// -------------------------------------------------
// Maintenance
      A     #U.Seq.Switch.Sw31;
      OPN   DB   500;
      =     DBX [AR2,P#0.0]; //"PStatD".U[#UnitNo].MTNC
// -------------------------------------------------
// CIP Required
// -------------------------------------------------
// CIP Active
// -------------------------------------------------
// CIP Clean
// -------------------------------------------------
// SIP Required
// -------------------------------------------------
// SIP Active
// -------------------------------------------------
// SIP Clean
// -------------------------------------------------
// Full
      A     DB135.DBX   26.2;
      OPN   DB   500;
      =     DBX [AR2,P#0.7]; //"PStatD".U[#UnitNo].FULL
// -------------------------------------------------
// Filling
      A     DB135.DBX   26.1;
      OPN   DB   500;
      =     DBX [AR2,P#1.0]; //"PStatD".U[#UnitNo].FILL
// -------------------------------------------------
// Ready For Filling
      A     DB135.DBX   26.0;
      OPN   DB   500;
      =     DBX [AR2,P#1.1]; //"PStatD".U[#UnitNo].RFFI
// -------------------------------------------------
// Empty
      A     DB135.DBX   26.5;
      OPN   DB   500;
      =     DBX [AR2,P#1.2]; //"PStatD".U[#UnitNo].EMTY
// -------------------------------------------------
// Emptying
      A     DB135.DBX   26.4;
      OPN   DB   500;
      =     DBX [AR2,P#1.3]; //"PStatD".U[#UnitNo].EMTI
// -------------------------------------------------
// Ready For Emptying
      A     DB135.DBX   26.3;
      OPN   DB   500;
      =     DBX [AR2,P#1.4]; //"PStatD".U[#UnitNo].RFEM
// -------------------------------------------------
// Reserved
//      A     #ComXYZ
//      OPN   "PStatD"
//      =     DBX [AR2,P#1.5]             //"PStatD".U[#UnitNo].RESV
// -------------------------------------------------
// Production
// -------------------------------------------------
// Used

// -------------------------------------------------
// PStat Function Call

      CALL FC   500 (
           UnitNo                   := #UnitNo,
           PStatModVal              := DB235.DBD  234);

NETWORK
TITLE =Unit Hold Request and Messages

      SET   ;

// ---------------------------------------------------------------------------
// Set unit to "hold" if maintenance
      AN    #U.Seq.Switch.Sw31; // maintenance !
      JC    NCO1;
      S     M    120.3;
      L     998; // "Unit in maintenance !"
      T     MD    90;

// ---------------------------------------------------------------------------
// Set unit to "hold" if emergency stop
NCO1: A     #EStopOK;
      JC    NCO2;
      S     M    120.3;
      L     999; // "Emergency stop !"
      T     MD    90;
NCO2: NOP   0;


// ---------------------------------------------------------------------------
// Check Partner
      AN    #ComSRC;
      O(    ;
      AN    DB135.DBX  314.3;
      AN    DB135.DBX  314.4;
      )     ;
      AN    #U.Seq.Step0;
      AN    #CIP;
      JCN   NC03;
      L     904; // "Source Not Ready!
      T     MD    90;
NC03: NOP   0;


      AN    DB135.DBX  266.0; // Water Tank Ready
      AN    DB135.DBX  266.1;
      AN    #ComDST;
      A     #S2I.SFM10.I00;
      AN    #U.Seq.Step0;
      AN    #U.Seq.PO.B22;
      AN    #U.Seq.PO.B3;
      AN    #CIP;
      JCN   NC04;
      L     903; // Destination not Ready
      T     MD    90;
NC04: NOP   0;



END_FUNCTION_BLOCK

FUNCTION_BLOCK FB 133
TITLE =C03: Local Well Transfer x
AUTHOR : Woermann
FAMILY : BOTEC_F1
NAME : C03E
VERSION : 1.2
CODE_VERSION1


VAR
  U : UDT 131;
END_VAR
VAR_TEMP
  CIP : BOOL ;	//CIP active
  UNIM : BOOL ;	//Unit Not In Maintenance
  GenRel : BOOL ;	//general OK (emergency and maintenance OK)
  EStopOK : BOOL ;	//emergency OK
  UnitNo : INT ;	//unit number
  xTmp : BOOL ;	//Temporary Bool
  iTmp : INT ;	//Temporary INT
  rTmp : REAL ;	//Temporary REAL
  dTmp : DINT ;	//Temporary DINT (free for general use)
  RetValInt : INT ;	//return value
  ComCIP1 : BOOL ;	//CIP1 in use
  ComCIP3 : BOOL ;	//CIP3 in use
END_VAR
BEGIN
NETWORK
TITLE =General

      SET   ;
// Simulation ---------------------------------------------------------------
      A     #U.Seq.User.Bit63;
      CC    FB   139; // "C03Sim"
      A     #U.Seq.Sim;
      =     #U.Seq.User.Bit63; //Help bit for simulation

// get unit number ----------------------------------------------------------
      L     MB   112;
      T     #UnitNo;

// CIP ----------------------------------------------------------------------
      L     #U.Seq.ProgNo;
      L     0;
      <D    ;
      =     #CIP;

// emergency OK -------------------------------------------------------------
      A     DB135.DBX   27.0; //Emergency Stop OK
      =     #EStopOK;

// Write Unit in Maintenance ------------------------------------------------

      AN    #U.Seq.Switch.Sw31;
      =     #UNIM;

// emergency and maintenance OK ---------------------------------------------
      A     #EStopOK;
      A     #UNIM;
      =     #GenRel;

// communication ------------------------------------------------------------
      UC    FB   135; // C03Com

NETWORK
TITLE =Analog Inputs

      NOP   0;

// ----------------------------------------------------------
// U31_AnI001 J6F_Druck
// ----------------------------------------------------------
      L     #U.Seq.SFM[63].Sp; // !!! insert correct SFM !!!
      T     DB233.DBD  238;

      SET   ;
      =     DB233.DBX  141.5;

// ----------------------------------------------------------
// QI_CO2_J6F_PH
// ----------------------------------------------------------
      L     #U.Seq.SFM[15].Sp;
      T     DB233.DBD  358;

      SET   ;
      =     DB233.DBX  261.5;

// ----------------------------------------------------------
// U31_AnI003 spare
// ----------------------------------------------------------
      L     #U.Seq.SFM[63].Sp; // !!! insert correct SFM !!!
      T     DB233.DBD  478;

      SET   ;
      =     DB233.DBX  381.5;

NETWORK
TITLE =Universal Value

      NOP   0;

// ----------------------------------------------------------
// unv001 Process Status
// ----------------------------------------------------------
// process value to UnV
//      L     0.000000e+000
//      T     "C03UnVD".unv001.ValExt

// ----------------------------------------------------------
// unv002 Universal Value 02
// ----------------------------------------------------------
// process value to UnV
//      L     0.000000e+000
//      T     "C03UnVD".unv002.ValExt

// ----------------------------------------------------------
// unv003 Universal Value 03
// ----------------------------------------------------------
// process value to UnV
//      L     0.000000e+000
//      T     "C03UnVD".unv003.ValExt

// ----------------------------------------------------------
// unv004 Universal Value 04
// ----------------------------------------------------------
// process value to UnV
//      L     0.000000e+000
//      T     "C03UnVD".unv004.ValExt

NETWORK
TITLE =Special Input

      NOP   0;

// ----------------------------------------------------------
// U31_SpI001 spare
// ----------------------------------------------------------
      CLR   ; // Only used in one well?
      =     DB231.DBX   81.4;
      =     DB231.DBX   81.5;

// ----------------------------------------------------------
// U31_SpI002 spare
// ----------------------------------------------------------
      CLR   ; // Only used in one well?
      =     DB231.DBX  141.4;
      =     DB231.DBX  141.5;

// ----------------------------------------------------------
// U31_SpI003 spare
// ----------------------------------------------------------
      CLR   ; // Only used in one well?
      =     DB231.DBX  201.4;
      =     DB231.DBX  201.5;

NETWORK
TITLE =Messages

      NOP   0;

// ----------------------------------------------------------
// msg001 Message 01
// ----------------------------------------------------------
      SET   ;
      R     DB237.DBX   80.7;
      =     DB237.DBX   81.4;

      CLR   ;
      =     DB237.DBX   82.7;

// ----------------------------------------------------------
// msg002 Message 02
// ----------------------------------------------------------
      SET   ;
      R     DB237.DBX  140.7;
      =     DB237.DBX  141.4;

      CLR   ;
      =     DB237.DBX  142.7;

// ----------------------------------------------------------
// msg003 Message 03
// ----------------------------------------------------------
      SET   ;
      R     DB237.DBX  200.7;
      =     DB237.DBX  201.4;

      CLR   ;
      =     DB237.DBX  202.7;

NETWORK
TITLE =PID controller
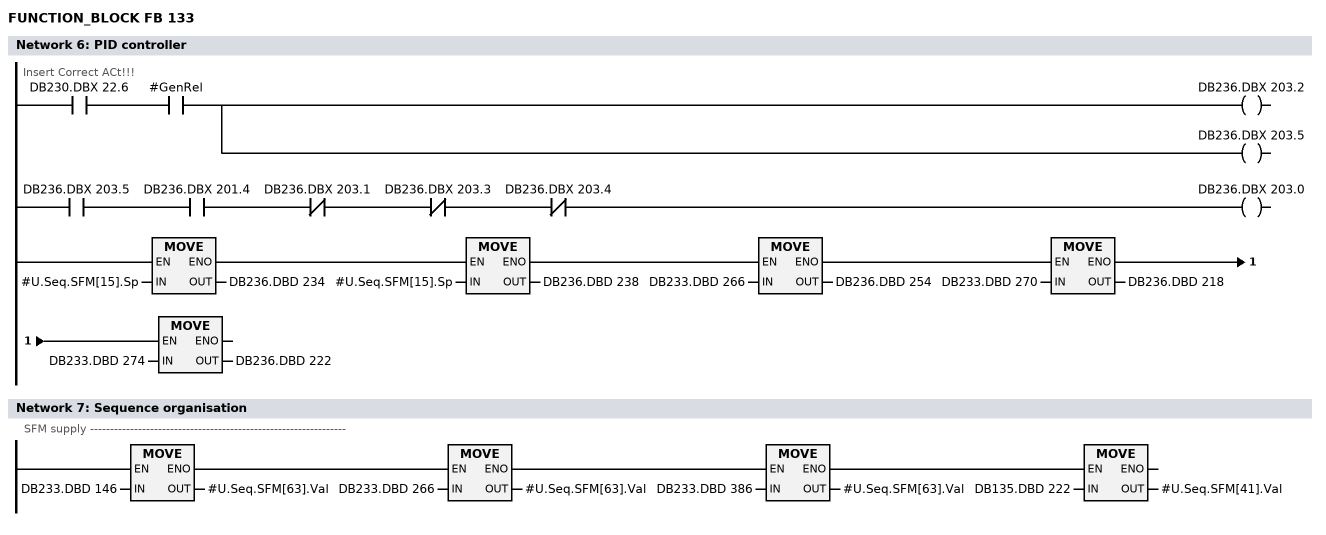

      NOP   0;

// ----------------------------------------------------------
// CO2J6FRV1 CO2 J6F RV1
// ----------------------------------------------------------
// starting value -----------------------
      A     DB230.DBX   22.6; // Insert Correct ACt!!!
      A     #GenRel;
      =     DB236.DBX  203.2;
      =     DB236.DBX  203.5;

// enable alarm -------------------------
      A     DB236.DBX  203.5;
      A     DB236.DBX  201.4;
      AN    DB236.DBX  203.1;
      AN    DB236.DBX  203.3;
      AN    DB236.DBX  203.4;
      =     DB236.DBX  203.0;

// setpoint to controller ---------------
      L     #U.Seq.SFM[15].Sp; // pH
      T     DB236.DBD  234;

// static value to controller ----------
      L     #U.Seq.SFM[15].Sp; //  pH
      T     DB236.DBD  238;

// process value to controller ----------
      L     DB233.DBD  266;
      T     DB236.DBD  254;

// low/high value to controller ---------
      L     DB233.DBD  270;
      T     DB236.DBD  218;

      L     DB233.DBD  274;
      T     DB236.DBD  222;

NETWORK
TITLE =Sequence organisation
//
// SFM supply ----------------------------------------------------------------

// analog value to SFM J6F_Druck -----------------------
      L     DB233.DBD  146;
      T     #U.Seq.SFM[63].Val;

// analog value to SFM QI_CO2_J6F_PH -------------------
      L     DB233.DBD  266;
      T     #U.Seq.SFM[63].Val; // !!! insert correct SFM !!!

// analog value to SFM spare -----------------------
      L     DB233.DBD  386;
      T     #U.Seq.SFM[63].Val; // !!! insert correct SFM !!!


// Amount from Well PLC04
      L     DB135.DBD  222;
      T     #U.Seq.SFM[41].Val;


NETWORK
TITLE =Auto / Manual

      SET   ;
      AN    M    122.2;
      JC    MODE;
      AN    M    120.1;

// assign actuator mode
      AN    M    120.1;
      =     DB230.DBX  105.4;
      =     DB230.DBX  185.4;
      =     DB230.DBX  265.4;

// assign PID mode
      S     DB236.DBX  201.4;
      S     DB236.DBX  201.5;

MODE: SET   ;

NETWORK
TITLE =C03_Act001 spare
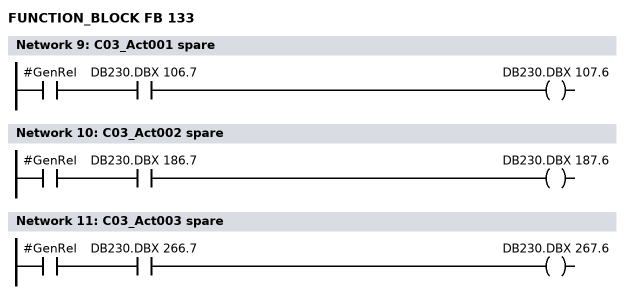

      A     #GenRel;
      A     DB230.DBX  106.7;
      =     DB230.DBX  107.6;
NETWORK
TITLE =C03_Act002 spare

      A     #GenRel;
      A     DB230.DBX  186.7;
      =     DB230.DBX  187.6;
NETWORK
TITLE =C03_Act003 spare

      A     #GenRel;
      A     DB230.DBX  266.7;
      =     DB230.DBX  267.6;
END_FUNCTION_BLOCK

FUNCTION_BLOCK FB 135
TITLE =C03: Local Well Transfer x
AUTHOR : Woermann
FAMILY : BOTEC_F1
NAME : C03Comm
VERSION : 0.1
CODE_VERSION1


VAR
  U : UDT 131;
END_VAR
VAR_TEMP
  iRetVal : INT ;	//return value as integer
  wRetVal : WORD ;	//return value as word
  Run : BOOL ;	//Unit in "RUN" mode
  EStopOK : BOOL ;	//Emergency Stop OK
  CIP : BOOL ;	//CIP Program Selected
  ComCIP : BOOL ;	//Communication with CIP Active
  xTmp : BOOL ;	//Temporary BOOL (free for general use)
  iTmp : INT ;	//Temporary INT (free for general use)
  rTmp : REAL ;	//Temporary REAL (free for general use)
  dTmp : DINT ;	//Temporary DINT (free for general use)
  UnitNo : INT ;	//Unit Number
  EquipmentID : INT ;	//Equipment ID
  Prid : DINT ;	//Process ID
  SFM36 : STRUCT 	//CIP Pump Mode
   I00 : BOOL ;	// Off
   I01 : BOOL ;	// Flow
   I02 : BOOL ;	// Pressure
   I03 : BOOL ;	// Fix Speed
   I04 : BOOL ;
   I05 : BOOL ;
   I06 : BOOL ;
   I07 : BOOL ;
   I08 : BOOL ;
   I09 : BOOL ;
   I10 : BOOL ;
   I11 : BOOL ;
   I12 : BOOL ;
   I13 : BOOL ;
   I14 : BOOL ;
   I15 : BOOL ;
   I16 : BOOL ;
   I17 : BOOL ;
   I18 : BOOL ;
   I19 : BOOL ;
   I20 : BOOL ;
   I21 : BOOL ;
   I22 : BOOL ;
   I23 : BOOL ;
   I24 : BOOL ;
   I25 : BOOL ;
   I26 : BOOL ;
   I27 : BOOL ;
   I28 : BOOL ;
   I29 : BOOL ;
   I30 : BOOL ;
   I31 : BOOL ;
  END_STRUCT ;
  iPLC : INT ;
  iUnit : INT ;
  rUnitNo : REAL ;
  DSTUnit : INT ;	//Destination Unit
END_VAR
BEGIN
NETWORK
TITLE =general

      SET   ;

// unit & equipment number ---------------------------------------------------
      L     #U.Seq.UnitNo;
      T     #UnitNo;

      L     DB135.DBW   14;
      L     1000;
      *I    ;
      L     #UnitNo;
      +I    ;
      T     #EquipmentID;

// CIP ----------------------------------------------------------------------
      L     DB135.DBW   18;
      L     0;
      <I    ;
      =     #CIP;

// Communicating Units-------------------------------------------------------
      L     DB135.DBD   10;
      L     DB135.DBD  106;
      ==D   ;
      =     #ComCIP;

// emergency OK -------------------------------------------------------------
      A     DB135.DBX   75.0; //General Emergency Stop OK
      =     #EStopOK;

NETWORK
TITLE =read other unit's data

      SET   ;

// ... General Unit ----------/
      CALL SFC   20 (
           SRCBLK                   := DB1995.Own,
           RET_VAL                  := #iTmp,
           DSTBLK                   := DB135.GEN);

// ... CIP Unit ------------- /

      CALL FC   563 (
           ActReq                   := M    101.0,
           PLCNo                    := 3,
           SourceUnitNo             := 91,
           IsTUnit                  := FALSE,
           DstComDRec               := DB135.CIP,
           RET_VAL                  := #wRetVal);

//----------------------------------------
// Communication Water Tank
//----------------------------------------
// Current Tank ----------------------------
      CALL FC   950 (
           EquipmentNo              := #U.Seq.SFM[10].Sp,
           PLCNo                    := #iPLC,
           UnitNo                   := #iUnit);

      L     #U.Seq.SFM[10].Sp;
      L     0.000000e+000;
      >R    ;
      JCN   N201;

      CALL FC   563 (
           ActReq                   := M    101.0,
           PLCNo                    := #iPLC,
           SourceUnitNo             := #iUnit,
           IsTUnit                  := FALSE,
           DstComDRec               := DB135.DST,
           RET_VAL                  := #wRetVal);
      JU    N2x1;
N201: NOP   0;
      L     0;
      T     #rTmp;
      CALL SFC   21 (
           BVAL                     := #rTmp,
           RET_VAL                  := #iTmp,
           BLK                      := DB135.DST);
N2x1: NOP   0;
// Priority 1 -----------------------------
      CALL FC   950 (
           EquipmentNo              := #U.Seq.SFM[11].Sp,
           PLCNo                    := #iPLC,
           UnitNo                   := #iUnit);

      L     #U.Seq.SFM[11].Sp;
      L     0.000000e+000;
      >R    ;
      JCN   N202;

      CALL FC   563 (
           ActReq                   := M    101.0,
           PLCNo                    := #iPLC,
           SourceUnitNo             := #iUnit,
           IsTUnit                  := FALSE,
           DstComDRec               := DB135.DST1,
           RET_VAL                  := #wRetVal);
      JU    N2x2;
N202: NOP   0;
      L     0;
      T     #rTmp;
      CALL SFC   21 (
           BVAL                     := #rTmp,
           RET_VAL                  := #iTmp,
           BLK                      := DB135.DST1);
N2x2: NOP   0;

// Priority 2 ----------------------------
      CALL FC   950 (
           EquipmentNo              := #U.Seq.SFM[12].Sp,
           PLCNo                    := #iPLC,
           UnitNo                   := #iUnit);

      L     #U.Seq.SFM[12].Sp;
      L     0.000000e+000;
      >R    ;
      JCN   N203;

      CALL FC   563 (
           ActReq                   := M    101.0,
           PLCNo                    := #iPLC,
           SourceUnitNo             := #iUnit,
           IsTUnit                  := FALSE,
           DstComDRec               := DB135.DST2,
           RET_VAL                  := #wRetVal);
      JU    N2x3;
N203: NOP   0;
      L     0;
      T     #rTmp;
      CALL SFC   21 (
           BVAL                     := #rTmp,
           RET_VAL                  := #iTmp,
           BLK                      := DB135.DST2);
N2x3: NOP   0;

// Priority 3 ----------------------------
      CALL FC   950 (
           EquipmentNo              := #U.Seq.SFM[13].Sp,
           PLCNo                    := #iPLC,
           UnitNo                   := #iUnit);

      L     #U.Seq.SFM[13].Sp;
      L     0.000000e+000;
      >R    ;
      JCN   N204;

      CALL FC   563 (
           ActReq                   := M    101.0,
           PLCNo                    := #iPLC,
           SourceUnitNo             := #iUnit,
           IsTUnit                  := FALSE,
           DstComDRec               := DB135.DST3,
           RET_VAL                  := #wRetVal);
      JU    N2x4;
N204: NOP   0;
      L     0;
      T     #rTmp;
      CALL SFC   21 (
           BVAL                     := #rTmp,
           RET_VAL                  := #iTmp,
           BLK                      := DB135.DST3);
N2x4: NOP   0;

//----------------------------------------
// Communication Water Treatment
//----------------------------------------
      L     21;
      L     DB135.DBW   16;
      ==I   ;
      JCN   WTR2;
      CALL FC   563 (
           ActReq                   := M    101.0,
           PLCNo                    := DB135.DBW   14,
           SourceUnitNo             := 38,
           IsTUnit                  := FALSE,
           DstComDRec               := DB135.PARTNER,
           RET_VAL                  := #wRetVal);
WTR2: L     22;
      ==I   ;
      JCN   NWTR;
      CALL FC   563 (
           ActReq                   := M    101.0,
           PLCNo                    := DB135.DBW   14,
           SourceUnitNo             := 39,
           IsTUnit                  := FALSE,
           DstComDRec               := DB135.PARTNER,
           RET_VAL                  := #wRetVal);

NWTR: NOP   0;

//----------------------------------------
// Communication Local Wells
//----------------------------------------
      L     #U.Seq.SFM[14].Sp; // Source
      T     #rTmp;

      CALL FC   950 (
           EquipmentNo              := #rTmp,
           PLCNo                    := #iPLC,
           UnitNo                   := #iUnit);

      L     #iUnit;
      L     1;
      ==I   ;
      JCN   U001;
      CALL SFC   20 (
           SRCBLK                   := DB1995.P04U001,
           RET_VAL                  := #iTmp,
           DSTBLK                   := DB135.SRC);
U001: NOP   0;

      L     #iUnit;
      L     2;
      ==I   ;
      JCN   U002;
      CALL SFC   20 (
           SRCBLK                   := DB1995.P04U002,
           RET_VAL                  := #iTmp,
           DSTBLK                   := DB135.SRC);
U002: NOP   0;

      L     #iUnit;
      L     3;
      ==I   ;
      JCN   U003;
      CALL SFC   20 (
           SRCBLK                   := DB1995.P04U003,
           RET_VAL                  := #iTmp,
           DSTBLK                   := DB135.SRC);
U003: NOP   0;

      L     #iUnit;
      L     4;
      ==I   ;
      JCN   U004;
      CALL SFC   20 (
           SRCBLK                   := DB1995.P04U004,
           RET_VAL                  := #iTmp,
           DSTBLK                   := DB135.SRC);
U004: NOP   0;

// Plan ----------------------------
      L     #UnitNo;
      L     100;
      +I    ;
      T     #iUnit;

      CALL FC   563 (
           ActReq                   := M    101.0,
           PLCNo                    := 3,
           SourceUnitNo             := #iUnit,
           IsTUnit                  := FALSE,
           DstComDRec               := DB135.PLN,
           RET_VAL                  := #wRetVal);

NETWORK
TITLE =external releases

      SET   ;
      =     DB230.DBX  106.7;
      =     DB230.DBX  186.7;
      =     DB230.DBX  266.7;

NETWORK
TITLE =write own unit data

      SET   ;
//-- CIP Communication ---------------------------------------
      AN    #U.Seq.Step0;
      AN    #U.Seq.PO.B30; // CIP Active (Slave)
      A     #ComCIP;
      JCN   NCIP;
//Conductivity CIP Return
      L     DB135.DBD  150;
      T     #U.Seq.SFM[32].Val;

//Temperature CIP Return
      L     DB135.DBD  146;
      T     #U.Seq.SFM[30].Val;

//CIP Prerun Pump SP

      CALL FC    45 (
           SFM                      := #U.Seq.SFM[36].Sp,
           Indexes                  := #SFM36);


      L     0.000000e+000;
      A     #SFM36.I01;
      =     DB135.DBX  171.7;
      JCN   pfc;
      L     #U.Seq.SFM[34].Sp;
pfc:  NOP   0;
      A     #SFM36.I02;
      =     DB135.DBX  172.0;
      JCN   ppc;
      L     #U.Seq.SFM[35].Sp;
ppc:  NOP   0;
      A     #SFM36.I03;
      =     DB135.DBX  171.6;
      JCN   pxc;
      L     #U.Seq.SFM[29].Sp;
pxc:  NOP   0;
      T     DB135.DBD  182;

//CIP Return
      L     #U.Seq.SFM[28].Sp;
      T     DB135.DBD  186;
      L     DB135.DBD  138;
      T     #U.Seq.SFM[28].Val;

//CIP Prerun
      L     #U.Seq.SFM[27].Sp;
      T     DB135.DBD  190;
      L     DB135.DBD  142;
      T     #U.Seq.SFM[27].Val;

// Write Own Data to CIP
      L     DB135.DBD   10;
      T     DB135.DBD  154;

      L     DB135.DBW   14;
      T     DB135.DBW  158;

      L     DB135.DBW   16;
      T     DB135.DBW  160;

      L     DB135.DBW   18;
      T     DB135.DBW  162;

      L     DB135.DBW   20;
      T     DB135.DBW  164;

      L     DB135.DBW   22;
      T     DB135.DBW  166;

      A     DB135.DBX   24.0;
      =     DB135.DBX  168.0;

      A     DB135.DBX   24.1;
      =     DB135.DBX  168.1;

      A     DB135.DBX   24.2;
      =     DB135.DBX  168.2;

      A     DB135.DBX   24.3;
      =     DB135.DBX  168.3;

      A     DB135.DBX   24.4;
      =     DB135.DBX  168.4;

      A     DB135.DBX   24.5;
      =     DB135.DBX  168.5;

      A     DB135.DBX   24.6;
      =     DB135.DBX  168.6;

      A     DB135.DBX   24.7;
      =     DB135.DBX  168.7;

// Copy Data to CIP
      CALL SFC   20 (
           SRCBLK                   := DB135.ToCIP,
           RET_VAL                  := #iRetVal,
           DSTBLK                   := DB135.ToCIP);

NCIP: NOP   0;

//Empty Signal
//A     "C03SpID".SpI.Sig //!!!! Insert correct Empty Signal !!!
      CLR   ;
      =     DB135.DBX   26.5;

//Full Signal
//A     "C03SpID".SpI.Sig //!!!! Insert correct Full Signal !!!
      CLR   ;
      =     DB135.DBX   26.2;

//CIP Program Selected
      A     #CIP;
      =     DB135.DBX   27.1;

// Emergency Stop
      A     #EStopOK; //If needed add or replace with own SpI
      =     DB135.DBX   27.0; //Emergency Stop OK

      L     #U.Seq.SFM[42].Sp; // Material
      T     DB135.DBD   30;

      L     DB135.DBD  326;
      T     #U.Seq.User.Real3;

//----------------------------------------
// Communication Water Tank
//----------------------------------------


      L     #U.Seq.SFM[10].Sp; // Current Tank
      T     DB135.DBD   34;

      L     #U.Seq.SFM[11].Sp; // Tank Priority 1
      T     DB135.DBD   38;

      L     #U.Seq.SFM[12].Sp; // Tank Priority 2
      T     DB135.DBD   42;

      L     #U.Seq.SFM[13].Sp; // Tank Priority 3
      T     DB135.DBD   46;

      L     #U.Seq.SFM[14].Sp; // Source
      T     DB135.DBD   50;

NETWORK
TITLE = read from other unit data




END_FUNCTION_BLOCK

FUNCTION_BLOCK FB 139
TITLE =C03: Local Well Transfer x
AUTHOR : Woermann
FAMILY : BOTEC_F1
NAME : C03Sim
VERSION : 0.1
CODE_VERSION1


VAR
  U : UDT 131;
END_VAR
VAR_TEMP
  CIP : BOOL ;	//CIP active
  xTmp : BOOL ;	//Temporary BOOL (free for general use)
  iTmp : INT ;	//Temporary INT (free for general use)
  rTmp : REAL ;	//Temporary REAL (free for general use)
  UnitNo : INT ;	//Unit Number
END_VAR
BEGIN
NETWORK
TITLE =General

      SET   ;
// get unit number ----------------------------------------------------------
      L     #U.Seq.UnitNo;
      T     #UnitNo;

// CIP ----------------------------------------------------------------------
      L     MW   114;
      L     0;
      <D    ;
      =     #CIP;

NETWORK
TITLE =Actuator

      A     #U.Seq.Sim;
      =     DB230.DBX  105.3;
      =     DB230.DBX  185.3;
      =     DB230.DBX  265.3;


NETWORK
TITLE =Special Input

      A     #U.Seq.Sim;
      =     DB231.DBX   81.3;
      =     DB231.DBX  141.3;
      =     DB231.DBX  201.3;

NETWORK
TITLE =Counter

      A     #U.Seq.Sim;
      A     M    101.0;

NETWORK
TITLE =Analog Input

      A     #U.Seq.Sim;
      =     DB233.DBX  141.3;
      =     DB233.DBX  261.3;
      =     DB233.DBX  381.3;
NETWORK
TITLE =Universal Value
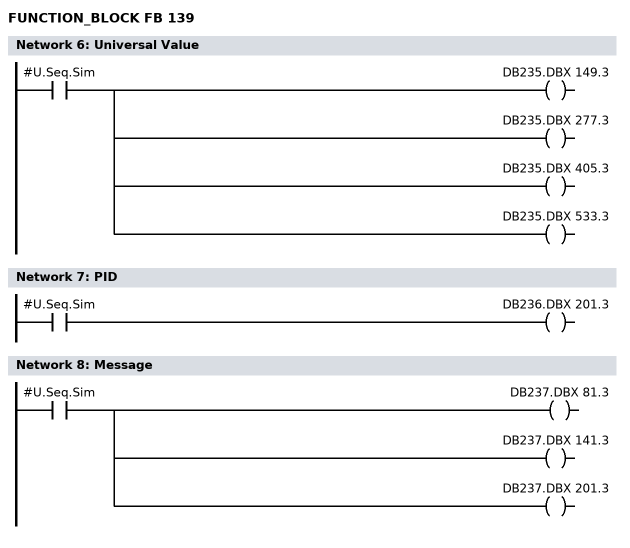

      A     #U.Seq.Sim;
      =     DB235.DBX  149.3;
      =     DB235.DBX  277.3;
      =     DB235.DBX  405.3;
      =     DB235.DBX  533.3;

NETWORK
TITLE =PID

      A     #U.Seq.Sim;
      =     DB236.DBX  201.3;

NETWORK
TITLE =Message

      A     #U.Seq.Sim;
      =     DB237.DBX   81.3;
      =     DB237.DBX  141.3;
      =     DB237.DBX  201.3;

NETWORK
TITLE =VLT

      A     #U.Seq.Sim;

END_FUNCTION_BLOCK

FUNCTION_BLOCK FB 141
TITLE =C04: Water Transfer Plant x
// NW  1 : phase and index evaluation
// NW  2 : phase  1: start position
// NW  3 : phase  3: Prerinse
// NW  4 : phase  4: Fill System
// NW  5 : phase  5: Transfer
// NW  6 : phase  8: Push Out
// NW  7 : phase 11: Postrinse
// NW  8 : phase 21: Prepare Line
// NW  9 : phase 22: Tank Selection
// NW 10 : phase 30: CIP Passive
// NW 11 : phase 31: CIP Start
// NW 12 : phase 32: CIP Push Out
// NW 13 : phase 34: CIP Rinsing
// NW 14 : phase 36: CIP Drain
// NW 15 : phase 40: CIP End
// NW 16 : end of sequence
// NW 17 : unit hold request
//SFM   Use                                 Datatype        UoM
//----+-------------------------------------------------------------------------
// 09 : Process Time                        Duration        min
// 40 : Density                             Value           kg/l
// 42 : Material                            Value
// 43 : Source                              Value
// 44 : Standby                             Value
AUTHOR : Woermann
NAME : C04Seq
VERSION : 0.1
CODE_VERSION1


VAR
  U : UDT 141;
END_VAR
VAR_TEMP
  CIP : BOOL ;	//CIP active
  ComCIP : BOOL ;	//Communication With CIP Active
  ComSRC : BOOL ;	//Communication With Well Transfer x
  RRel : BOOL ;	//Run Release
  EStopOK : BOOL ;	//emergency OK
  StepMax : BOOL ;	//StepMax (last) active
  SubStepMax : BOOL ;	//SubStepMax (last) active
  SubStepMaxD : BOOL ;	//SubStepMax (last) done
  ChkOK : BOOL ;	//SubStepMax (last) done
  xTmp : BOOL ;	//Temporary BOOL (free for general use)
  iTmp : INT ;	//Temporary INT (free for general use)
  dTmp : DINT ;	//Temporary DINT (free for general use)
  wTmp : WORD ;
  rTmp : REAL ;	//Temporary REAL (free for general use)
  dUnitNo : DINT ;	//Unit Number
  UnitNo : INT ;	//Unit Number
  EquipmentID : INT ;	//Equipment ID
  S2I : STRUCT 	//SFM to indexes
   SFM26 : STRUCT 	//CIP Step On Condition
    I00 : BOOL ;	//Please Select
    I01 : BOOL ;	//Conductivity High
    I02 : BOOL ;	//Conductivity Low
    I03 : BOOL ;	//Time
    I04 : BOOL ;	//Amount
    I05 : BOOL ;	//Temperature High
    I06 : BOOL ;	//Temperature Low
    I07 : BOOL ;
    I08 : BOOL ;
    I09 : BOOL ;
    I10 : BOOL ;
    I11 : BOOL ;
    I12 : BOOL ;
    I13 : BOOL ;
    I14 : BOOL ;
    I15 : BOOL ;
    I16 : BOOL ;
    I17 : BOOL ;
    I18 : BOOL ;
    I19 : BOOL ;
    I20 : BOOL ;
    I21 : BOOL ;
    I22 : BOOL ;
    I23 : BOOL ;
    I24 : BOOL ;
    I25 : BOOL ;
    I26 : BOOL ;
    I27 : BOOL ;
    I28 : BOOL ;
    I29 : BOOL ;
    I30 : BOOL ;
    I31 : BOOL ;
   END_STRUCT ;
   SFM27 : STRUCT 	//CIP Prerun
    I00 : BOOL ;	//None
    I01 : BOOL ;	//Recovered Water
    I02 : BOOL ;	//Caustic
    I03 : BOOL ;
    I04 : BOOL ;	//Acid
    I05 : BOOL ;
    I06 : BOOL ;
    I07 : BOOL ;
    I08 : BOOL ;
    I09 : BOOL ;
    I10 : BOOL ;
    I11 : BOOL ;
    I12 : BOOL ;	//Fresh Water
    I13 : BOOL ;	//Warm Water
    I14 : BOOL ;
    I15 : BOOL ;
    I16 : BOOL ;
    I17 : BOOL ;
    I18 : BOOL ;
    I19 : BOOL ;
    I20 : BOOL ;
    I21 : BOOL ;
    I22 : BOOL ;
    I23 : BOOL ;
    I24 : BOOL ;
    I25 : BOOL ;
    I26 : BOOL ;
    I27 : BOOL ;
    I28 : BOOL ;
    I29 : BOOL ;
    I30 : BOOL ;
    I31 : BOOL ;
   END_STRUCT ;
   SFM28 : STRUCT 	//CIP Return
    I00 : BOOL ;	//None
    I01 : BOOL ;	//Recovered Water
    I02 : BOOL ;	//Caustic
    I03 : BOOL ;
    I04 : BOOL ;	//Acid
    I05 : BOOL ;
    I06 : BOOL ;
    I07 : BOOL ;
    I08 : BOOL ;
    I09 : BOOL ;
    I10 : BOOL ;
    I11 : BOOL ;
    I12 : BOOL ;	//Fresh Water
    I13 : BOOL ;	//Warm Water
    I14 : BOOL ;
    I15 : BOOL ;	//Drain
    I16 : BOOL ;
    I17 : BOOL ;
    I18 : BOOL ;
    I19 : BOOL ;
    I20 : BOOL ;
    I21 : BOOL ;
    I22 : BOOL ;
    I23 : BOOL ;
    I24 : BOOL ;
    I25 : BOOL ;
    I26 : BOOL ;
    I27 : BOOL ;
    I28 : BOOL ;
    I29 : BOOL ;
    I30 : BOOL ;
    I31 : BOOL ;
   END_STRUCT ;
   SFM37 : STRUCT 	//CIP Pump Mode
    I00 : BOOL ;	//Off
    I01 : BOOL ;	//Flow
    I02 : BOOL ;	//Pressure
    I03 : BOOL ;	//Fix Speed
    I04 : BOOL ;
    I05 : BOOL ;
    I06 : BOOL ;
    I07 : BOOL ;
    I08 : BOOL ;
    I09 : BOOL ;
    I10 : BOOL ;
    I11 : BOOL ;
    I12 : BOOL ;
    I13 : BOOL ;
    I14 : BOOL ;
    I15 : BOOL ;
    I16 : BOOL ;
    I17 : BOOL ;
    I18 : BOOL ;
    I19 : BOOL ;
    I20 : BOOL ;
    I21 : BOOL ;
    I22 : BOOL ;
    I23 : BOOL ;
    I24 : BOOL ;
    I25 : BOOL ;
    I26 : BOOL ;
    I27 : BOOL ;
    I28 : BOOL ;
    I29 : BOOL ;
    I30 : BOOL ;
    I31 : BOOL ;
   END_STRUCT ;
   SFM31 : STRUCT 	//CIP Distribution Circuit No
    I00 : BOOL ;	//Please Select
    I01 : BOOL ;	//Auto Select
    I02 : BOOL ;
    I03 : BOOL ;
    I04 : BOOL ;
    I05 : BOOL ;
    I06 : BOOL ;
    I07 : BOOL ;
    I08 : BOOL ;
    I09 : BOOL ;
    I10 : BOOL ;
    I11 : BOOL ;
    I12 : BOOL ;
    I13 : BOOL ;
    I14 : BOOL ;
    I15 : BOOL ;
    I16 : BOOL ;
    I17 : BOOL ;
    I18 : BOOL ;
    I19 : BOOL ;
    I20 : BOOL ;
    I21 : BOOL ;
    I22 : BOOL ;
    I23 : BOOL ;
    I24 : BOOL ;
    I25 : BOOL ;
    I26 : BOOL ;
    I27 : BOOL ;
    I28 : BOOL ;
    I29 : BOOL ;
    I30 : BOOL ;
    I31 : BOOL ;
   END_STRUCT ;
   SFM39 : STRUCT 	//Q-Status
    I00 : BOOL ;	//Please select
    I01 : BOOL ;	//released
    I02 : BOOL ;
    I03 : BOOL ;
    I04 : BOOL ;
    I05 : BOOL ;
    I06 : BOOL ;	//Ignore
    I07 : BOOL ;
    I08 : BOOL ;
    I09 : BOOL ;	//locked
    I10 : BOOL ;
    I11 : BOOL ;
    I12 : BOOL ;
    I13 : BOOL ;
    I14 : BOOL ;
    I15 : BOOL ;
    I16 : BOOL ;
    I17 : BOOL ;
    I18 : BOOL ;
    I19 : BOOL ;
    I20 : BOOL ;
    I21 : BOOL ;
    I22 : BOOL ;
    I23 : BOOL ;
    I24 : BOOL ;
    I25 : BOOL ;
    I26 : BOOL ;
    I27 : BOOL ;
    I28 : BOOL ;
    I29 : BOOL ;
    I30 : BOOL ;
    I31 : BOOL ;
   END_STRUCT ;
   SFM10 : STRUCT 	//Current Tank
    I00 : BOOL ;	//Please Select
    I01 : BOOL ;	//Water Tank 1
    I02 : BOOL ;	//Water Tank 2
    I03 : BOOL ;	//Water Tank 2
    I04 : BOOL ;	//Water Tank 3
    I05 : BOOL ;	//Water Tank 4
    I06 : BOOL ;	//Water Tank 5
    I07 : BOOL ;	//Water Tank 6
    I08 : BOOL ;	//Water Tank 7
    I09 : BOOL ;	//Water Tank 8
    I10 : BOOL ;	//WAter Tank 9
    I11 : BOOL ;	//Water Tank 10
    I12 : BOOL ;	//Water Tank 11
    I13 : BOOL ;	//Water Tank 12
    I14 : BOOL ;	//Water Tank 13
    I15 : BOOL ;
    I16 : BOOL ;
    I17 : BOOL ;
    I18 : BOOL ;
    I19 : BOOL ;
    I20 : BOOL ;
    I21 : BOOL ;
    I22 : BOOL ;
    I23 : BOOL ;
    I24 : BOOL ;
    I25 : BOOL ;
    I26 : BOOL ;
    I27 : BOOL ;
    I28 : BOOL ;
    I29 : BOOL ;
    I30 : BOOL ;
    I31 : BOOL ;
   END_STRUCT ;
   SFM11 : STRUCT 	//1. Tank
    I00 : BOOL ;	//Please Select
    I01 : BOOL ;	//Water Tank 1
    I02 : BOOL ;	//Water Tank 2
    I03 : BOOL ;	//Water Tank 2
    I04 : BOOL ;	//Water Tank 3
    I05 : BOOL ;	//Water Tank 4
    I06 : BOOL ;	//Water Tank 5
    I07 : BOOL ;	//Water Tank 6
    I08 : BOOL ;	//Water Tank 7
    I09 : BOOL ;	//Water Tank 8
    I10 : BOOL ;	//WAter Tank 9
    I11 : BOOL ;	//Water Tank 10
    I12 : BOOL ;	//Water Tank 11
    I13 : BOOL ;	//Water Tank 12
    I14 : BOOL ;	//Water Tank 13
    I15 : BOOL ;
    I16 : BOOL ;
    I17 : BOOL ;
    I18 : BOOL ;
    I19 : BOOL ;
    I20 : BOOL ;
    I21 : BOOL ;
    I22 : BOOL ;
    I23 : BOOL ;
    I24 : BOOL ;
    I25 : BOOL ;
    I26 : BOOL ;
    I27 : BOOL ;
    I28 : BOOL ;
    I29 : BOOL ;
    I30 : BOOL ;
    I31 : BOOL ;
   END_STRUCT ;
   SFM12 : STRUCT 	//2. Tank
    I00 : BOOL ;	//Please Select
    I01 : BOOL ;	//Water Tank 1
    I02 : BOOL ;	//Water Tank 2
    I03 : BOOL ;	//Water Tank 2
    I04 : BOOL ;	//Water Tank 3
    I05 : BOOL ;	//Water Tank 4
    I06 : BOOL ;	//Water Tank 5
    I07 : BOOL ;	//Water Tank 6
    I08 : BOOL ;	//Water Tank 7
    I09 : BOOL ;	//Water Tank 8
    I10 : BOOL ;	//WAter Tank 9
    I11 : BOOL ;	//Water Tank 10
    I12 : BOOL ;	//Water Tank 11
    I13 : BOOL ;	//Water Tank 12
    I14 : BOOL ;	//Water Tank 13
    I15 : BOOL ;
    I16 : BOOL ;
    I17 : BOOL ;
    I18 : BOOL ;
    I19 : BOOL ;
    I20 : BOOL ;
    I21 : BOOL ;
    I22 : BOOL ;
    I23 : BOOL ;
    I24 : BOOL ;
    I25 : BOOL ;
    I26 : BOOL ;
    I27 : BOOL ;
    I28 : BOOL ;
    I29 : BOOL ;
    I30 : BOOL ;
    I31 : BOOL ;
   END_STRUCT ;
   SFM13 : STRUCT 	//3. Tank
    I00 : BOOL ;	//Please Select
    I01 : BOOL ;	//Water Tank 1
    I02 : BOOL ;	//Water Tank 2
    I03 : BOOL ;	//Water Tank 2
    I04 : BOOL ;	//Water Tank 3
    I05 : BOOL ;	//Water Tank 4
    I06 : BOOL ;	//Water Tank 5
    I07 : BOOL ;	//Water Tank 6
    I08 : BOOL ;	//Water Tank 7
    I09 : BOOL ;	//Water Tank 8
    I10 : BOOL ;	//WAter Tank 9
    I11 : BOOL ;	//Water Tank 10
    I12 : BOOL ;	//Water Tank 11
    I13 : BOOL ;	//Water Tank 12
    I14 : BOOL ;	//Water Tank 13
    I15 : BOOL ;
    I16 : BOOL ;
    I17 : BOOL ;
    I18 : BOOL ;
    I19 : BOOL ;
    I20 : BOOL ;
    I21 : BOOL ;
    I22 : BOOL ;
    I23 : BOOL ;
    I24 : BOOL ;
    I25 : BOOL ;
    I26 : BOOL ;
    I27 : BOOL ;
    I28 : BOOL ;
    I29 : BOOL ;
    I30 : BOOL ;
    I31 : BOOL ;
   END_STRUCT ;
   SFM14 : STRUCT 	//3. Tank
    I00 : BOOL ;	//Please Select
    I01 : BOOL ;	//Yes
    I02 : BOOL ;	//No
    I03 : BOOL ;
    I04 : BOOL ;
    I05 : BOOL ;
    I06 : BOOL ;
    I07 : BOOL ;
    I08 : BOOL ;
    I09 : BOOL ;
    I10 : BOOL ;
    I11 : BOOL ;
    I12 : BOOL ;
    I13 : BOOL ;
    I14 : BOOL ;
    I15 : BOOL ;
    I16 : BOOL ;
    I17 : BOOL ;
    I18 : BOOL ;
    I19 : BOOL ;
    I20 : BOOL ;
    I21 : BOOL ;
    I22 : BOOL ;
    I23 : BOOL ;
    I24 : BOOL ;
    I25 : BOOL ;
    I26 : BOOL ;
    I27 : BOOL ;
    I28 : BOOL ;
    I29 : BOOL ;
    I30 : BOOL ;
    I31 : BOOL ;
   END_STRUCT ;
   SFM18 : STRUCT 	//CIP Start / CIP Distribution Start
    I00 : BOOL ;	//Please Select
    I01 : BOOL ;	//CIP 1
    I02 : BOOL ;	//CIP 2
    I03 : BOOL ;	//CIP 3
    I04 : BOOL ;	//Auto Select
    I05 : BOOL ;
    I06 : BOOL ;
    I07 : BOOL ;
    I08 : BOOL ;
    I09 : BOOL ;
    I10 : BOOL ;
    I11 : BOOL ;
    I12 : BOOL ;
    I13 : BOOL ;
    I14 : BOOL ;
    I15 : BOOL ;
    I16 : BOOL ;
    I17 : BOOL ;
    I18 : BOOL ;
    I19 : BOOL ;
    I20 : BOOL ;
    I21 : BOOL ;
    I22 : BOOL ;
    I23 : BOOL ;
    I24 : BOOL ;
    I25 : BOOL ;
    I26 : BOOL ;
    I27 : BOOL ;
    I28 : BOOL ;
    I29 : BOOL ;
    I30 : BOOL ;
    I31 : BOOL ;
   END_STRUCT ;
   SFM24 : STRUCT 	//Confirm Connections
    I00 : BOOL ;	//Please Select
    I01 : BOOL ;	//Yes
    I02 : BOOL ;	//No
    I03 : BOOL ;
    I04 : BOOL ;
    I05 : BOOL ;
    I06 : BOOL ;
    I07 : BOOL ;
    I08 : BOOL ;
    I09 : BOOL ;
    I10 : BOOL ;
    I11 : BOOL ;
    I12 : BOOL ;
    I13 : BOOL ;
    I14 : BOOL ;
    I15 : BOOL ;
    I16 : BOOL ;
    I17 : BOOL ;
    I18 : BOOL ;
    I19 : BOOL ;
    I20 : BOOL ;
    I21 : BOOL ;
    I22 : BOOL ;
    I23 : BOOL ;
    I24 : BOOL ;
    I25 : BOOL ;
    I26 : BOOL ;
    I27 : BOOL ;
    I28 : BOOL ;
    I29 : BOOL ;
    I30 : BOOL ;
    I31 : BOOL ;
   END_STRUCT ;
  END_STRUCT ;
  ComDST : BOOL ;	//Communication Water Transfer to Packaging Plant
  ComCIPDist : BOOL ;	//Communication with CIP Distribution
  CurrSel : REAL ;	//Current Tank Selection SP
  comWTank1 : BOOL ;	//Communication Water Tank Priority 1
  comWTank2 : BOOL ;	//Communication Water Tank Priority 2
  comWTank3 : BOOL ;	//Communication Water Tank Priority 3
  RelInlet : BOOL ;
  ComCIP1 : BOOL ;	//Communication With CIP1
  ComCIP2 : BOOL ;	//Communication With CIP2
  ComCIP3 : BOOL ;	//Communication With CIP3
  Empty : BOOL ;
  ComDistCIP1 : BOOL ;	//Communication With CIP Distribution 1
  ComDistCIP2 : BOOL ;	//Communication With CIP Distribution 2
  ComDistCIP3 : BOOL ;	//Communication With CIP Distribution 3
  LineID : INT ;	// LineTank Com ID
END_VAR
BEGIN
NETWORK
TITLE = Phase and Index Evaluation

      CLR   ;
      =     #RRel;
      =     #xTmp;
      =     DB145.DBX   29.5;
      =     DB145.DBX   29.7;
      =     DB145.DBX  173.7;

      L     MB   112;
      L     43;
      -I    ;
      JL    LIDE;
      JU    ID43;
      JU    LIDE;
      JU    ID45;
      JU    LIDE;
      JU    ID47;
      JU    LIDE;
      JU    ID49;
      JU    ID50;
      JU    ID51;
      JU    ID52;
      JU    LIDE;
      JU    ID54;
      JU    LIDE;
      JU    ID56;
      JU    ID57;
      JU    ID58;
      JU    LIDE;
LIDE: L     0;
      JU    FIM1;
ID43: L     1;
      JU    FIM1;
ID45: L     2;
      JU    FIM1;
ID47: L     4;
      JU    FIM1;
ID49: L     8;
      JU    FIM1;
ID50: L     16;
      JU    FIM1;
ID51: L     32;
      JU    FIM1;
ID52: L     64;
      JU    FIM1;
ID54: L     128;
      JU    FIM1;
ID56: L     256;
      JU    FIM1;
ID57: L     512;
      JU    FIM1;
ID58: L     1024;
      JU    FIM1;
FIM1: NOP   0;
      T     #LineID;

// ---------------------------------------------------------------------------
// write max used SFM's (last SFM number + 1)
      L     60;
      T     #U.SFMQuant;

// ---------------------------------------------------------------------------
// unit & equipment number
      L     MB   112;
      T     #UnitNo;

      L     DB145.DBW   14;
      L     1000;
      *I    ;
      L     #UnitNo;
      +I    ;
      T     #EquipmentID;

// ---------------------------------------------------------------------------
// CIP active
      L     MW   114;
      L     0;
      <I    ;
      =     #CIP;

// ---------------------------------------------------------------------------
// communicating units
      L     MD   124;
      L     DB145.DBD  106;
      ==D   ;
      =     #ComCIP;

      L     MD   124;
      L     DB145.DBD  394;
      ==D   ;
      A     DB145.DBX  411.4;
      =     #ComCIPDist;

      L     DB145.DBW  400;
      L     94;
      ==I   ;
      =     #ComDistCIP1;

      L     DB145.DBW  400;
      L     95;
      ==I   ;
      =     #ComDistCIP2;

      L     DB145.DBW  400;
      L     96;
      ==I   ;
      =     #ComDistCIP3;

      L     DB145.DBW  112;
      L     91;
      ==I   ;
      =     #ComCIP1;

      L     DB145.DBW  112;
      L     92;
      ==I   ;
      =     #ComCIP2;

      L     DB145.DBW  112;
      L     93;
      ==I   ;
      =     #ComCIP3;


//---
      AN    M    120.7;
      =     #ComSRC;

      L     MD   124;
      L     DB145.DBD  442;
      ==D   ;
      =     #ComDST;

// ---------------------------------------------------------------------------
// process timer start
      SET   ;
      =     M    131.0;

// ---------------------------------------------------------------------------
// emergency OK
      A     DB145.DBX   27.0;
      =     #EStopOK;

// define last (Sub)Step active
      L     #U.Seq.StepMax;
      L     MW   104;
      ==I   ;
      =     #StepMax;

      L     #U.Seq.SubStepMax;
      L     MW   118;
      ==I   ;
      =     #SubStepMax;

      A     #SubStepMax;
      A     #U.Seq.SPD;
      AN    M    103.2;
      =     #SubStepMaxD;

// ---------------------------------------------------------------------------
// index evaluation: Current Tank
      CALL FC    45 (
           SFM                      := #U.Seq.SFM[10].Sp,
           Indexes                  := #S2I.SFM10);

// index evaluation: 1. Tank
      CALL FC    45 (
           SFM                      := #U.Seq.SFM[11].Sp,
           Indexes                  := #S2I.SFM11);

// index evaluation: 2. Tank
      CALL FC    45 (
           SFM                      := #U.Seq.SFM[12].Sp,
           Indexes                  := #S2I.SFM12);

// index evaluation: 3. Tank
      CALL FC    45 (
           SFM                      := #U.Seq.SFM[13].Sp,
           Indexes                  := #S2I.SFM13);

// index evaluation: Trap Filter
      CALL FC    45 (
           SFM                      := #U.Seq.SFM[14].Sp,
           Indexes                  := #S2I.SFM14);

// index evaluation: Q-Status
      CALL FC    45 (
           SFM                      := #U.Seq.SFM[39].Sp,
           Indexes                  := #S2I.SFM39);

// index evaluation: CIP Distribution Start
      CALL FC    45 (
           SFM                      := #U.Seq.SFM[18].Sp,
           Indexes                  := #S2I.SFM18);


// Tank Priority Selection
      CALL FC   779 (
           P1Sel                    := #U.Seq.SFM[11].Sp,
           P2Sel                    := #U.Seq.SFM[12].Sp,
           P3Sel                    := #U.Seq.SFM[13].Sp,
           P1Rel                    := DB145.DBX  267.3,
           P2Rel                    := DB145.DBX  315.3,
           P3Rel                    := DB145.DBX  363.3,
           CurrSel                  := #U.Seq.User.Real10);


// ---------------------------------------------------------------------------
// phase evaluation
      L     MW   108;
      JL    X0;
      JU    X0; // phase  0:
      JU    X1; // phase  1: start position
      JU    X0; // phase  2:
      JU    X3; // phase  3: Prerinse
      JU    X4; // phase  4: Fill System
      JU    X5; // phase  5: Transfer
      JU    X0; // phase  6:
      JU    X0; // phase  7:
      JU    X8; // phase  8: Push Out
      JU    X0; // phase  9:
      JU    X0; // phase 10:
      JU    X11; // phase 11: Postrinse
      JU    X0; // phase 12:
      JU    X0; // phase 13:
      JU    X0; // phase 14:
      JU    X0; // phase 15:
      JU    X0; // phase 16:
      JU    X0; // phase 17:
      JU    X0; // phase 18:
      JU    X19; // phase 19: Remove Filter Candles
      JU    X20; // phase 20: Replace Filter Candles
      JU    X21; // phase 21: Prepare Line
      JU    X22; // phase 22: Tank Selection
      JU    X0; // phase 23:
      JU    X0; // phase 24:
      JU    X0; // phase 25:
      JU    X0; // phase 26:
      JU    X0; // phase 27:
      JU    X0; // phase 28:
      JU    X0; // phase 29:
      JU    X30; // phase 30: CIP Active
      JU    X31; // phase 31: CIP Start
      JU    X32; // phase 32: CIP Prerun
      JU    X33; // phase 33: CIP Return
      JU    X34; // phase 34: CIP Rinsing
      JU    X35; // phase 35: CIP Emptying
      JU    X36; // phase 36: CIP Drain
      JU    X0; // phase 37:
      JU    X38; // phase 38: CIP Randvollstellung
      JU    X39; // phase 39: CIP Rinsing from RWT
      JU    X40; // phase 40: CIP End
X0:   SET   ;
      S     M    108.7; // Error unknown phase
      JU    COMM;
NETWORK
TITLE =phase 1: startposition

X1:   SET   ;

// ---------------------------------------------------------------------------
// general functions
// ---------------------------------------------------------------------------
// reset signals
      A     M    102.2;
      R     #U.Seq.Switch.Sw1;
      R     #U.Seq.Switch.Sw2;

      A     M    102.0;
      R     DB145.DBX   26.1;
      L     0;
      T     #U.Seq.SFM[10].Sp;
      T     #U.Seq.SFM[11].Sp;
      T     #U.Seq.SFM[12].Sp;
      T     #U.Seq.SFM[13].Sp;


      AN    M    102.0;
      =     M    161.0; // Reset Process Timer

      CALL FC   709 (// Reset "Simulation" And "Ignore"
           UnitNo                   := #UnitNo,// Of All Control Modules
           Enable                   := M    102.2);// At First Cycle of Startposition (Idle)

// ---------------------------------------------------------------------------
// start check --------------------------------------------------------------
      A     #CIP;
      JC    M010;

      CALL FC   140 (
           ChkType                  := 1,// production
           ChkOK                    := M    122.0);
      JU    COMM;

M010: CALL FC   140 (
           ChkType                  := 2,// CIP
           ChkOK                    := M    122.0);
      JU    COMM;

NETWORK
TITLE =phase 3: Prerinse
//SFM   Use                                 Datatype        UoM
//----+-------------------------------------------------------------------------
// 00 : Watch Dog Time                      Duration        min
// 20 : Flow                                Value           l/h
// 41 : Amount                              Value           kg
X3:   SET   ;
// ---------------------------------------------------------------------------
// General CM evaluation
      CALL FC   140 (
           ChkType                  := 3,
           ChkOK                    := #ChkOK);

      AN    #ChkOK;
      S     M    120.3;

// ---------------------------------------------------------------------------
// general functions
      AN    M    121.2;
      A     M    102.3;
      =     #RRel;

// ---------------------------------------------------------------------------
// messages
// ---------------------------------------------------------------------------
// timer & counter
      A     M    102.0;

// ---------------------------------------------------------------------------
// pause timer
// ---------------------------------------------------------------------------
// communication

// ---------------------------------------------------------------------------
// control modules
      A     M    102.3;

// ---------------------------------------------------------------------------
// transition condition
      A     #SubStepMaxD;
      =     M    102.1;

// subphase evaluation
      L     MW   110;
      JL    A300;
      JU    COMM; // subphase  0:
// ---------------------------------------------------------------------------
A300: SET   ;
      S     M    110.7; // Error unknown subphase
      JU    COMM;
NETWORK
TITLE =phase 4: Fill System
//SFM   Use                                 Datatype        UoM
//----+-------------------------------------------------------------------------
// 00 : Watch Dog Time                      Duration        min
// 20 : Flow                                Value           l/h
// 41 : Amount                              Value           kg
X4:   SET   ;
// ---------------------------------------------------------------------------
// General CM evaluation
      CALL FC   140 (
           ChkType                  := 3,
           ChkOK                    := #ChkOK);

      AN    #ChkOK;
      S     M    120.3;

// ---------------------------------------------------------------------------
// general functions
      AN    M    121.2;
      A     M    102.3;
      =     #RRel;

// ---------------------------------------------------------------------------
// messages
// ---------------------------------------------------------------------------
// timer & counter
      A     M    102.0;

// ---------------------------------------------------------------------------
// pause timer
// ---------------------------------------------------------------------------
// communication

// ---------------------------------------------------------------------------
// control modules
      A     M    102.3;

// ---------------------------------------------------------------------------
// transition condition
      A     #SubStepMaxD;
      =     M    102.1;

// subphase evaluation
      L     MW   110;
      JL    A400;
      JU    COMM; // subphase  0:
// ---------------------------------------------------------------------------
A400: SET   ;
      S     M    110.7; // Error unknown subphase
      JU    COMM;
NETWORK
TITLE =phase 5: Transfer
//SFM   Use                                 Datatype        UoM
//----+-------------------------------------------------------------------------
// 00 : Watch Dog Time                      Duration        min
// 20 : Flow                                Value           l/h
// 41 : Amount                              Value           kg
X5:   SET   ;
// ---------------------------------------------------------------------------
// General CM evaluation
      CALL FC   140 (
           ChkType                  := 3,
           ChkOK                    := #ChkOK);

      AN    #ChkOK;
      S     M    120.3;

// ---------------------------------------------------------------------------
// general functions
// ---------------------------------------------------------------------------
// messages
// ---------------------------------------------------------------------------
// timer & counter
      A     M    102.0;

// ---------------------------------------------------------------------------
// pause timer
// ---------------------------------------------------------------------------
// communication
// Communication Water Tank
      L     #LineID;
      L     DB145.DBD  242;
      AW    ;
      L     #LineID;
      ==I   ;
      AN    M    121.2;
      A     M    102.3;
      =     #RRel;

// Communication Water Tank
      A     M    103.3;
      =     DB145.DBX   26.1;

      A     DB145.DBX  218.4;
      A     #RRel;
      =     DB145.DBX   26.4;

// ---------------------------------------------------------------------------
// control modules
      A     M    102.3;

// ---------------------------------------------------------------------------
// transition condition
      CLR   ;
      =     M    102.1;

// ---------------------------------------------------------------------------
// ---------------------------------------------------------------------------
// subphase repeat function
      A     #SubStepMax;
      JCN   Y5;
      L     1;
      T     MW   116;
Y5:   SET   ;

// subphase evaluation
      L     MW   110;
      JL    A500;
      JU    COMM; // subphase  0:
      JU    A501; // subphase  1: Waiting
      JU    A502; // subphase  2: Active
      JU    A503; // subphase  3: Tank Change
// ---------------------------------------------------------------------------
A500: SET   ;
      S     M    110.7; // Error unknown subphase
      JU    COMM;

// subphase 1: Waiting
A501: SET   ;
      A     M    103.3;
      =     DB145.DBX   26.3; // Plant Comm
      =     DB145.DBX   26.0; // Tank Comm
// -------------------------------------------------
// subphase timer & counter
      A     M    103.0;

// -------------------------------------------------
// subphase actuator
      A     M    103.3;

// -------------------------------------------------
// subphase transition
      L     #U.Seq.User.Real10;
      L     #U.Seq.SFM[10].Sp;
      <>R   ;
      O     #S2I.SFM10.I00;
      =     #xTmp;

      A     #xTmp;
      O     DB145.DBX   26.4;
      =     M    103.1;
      JU    COMM;

// subphase 2: Active
A502: SET   ;


// -------------------------------------------------
// subphase timer & counter
      A     M    103.0;

// -------------------------------------------------
// subphase actuator
      A     #S2I.SFM14.I01;
      A     M    103.3;
      =     DB240.DBX  188.0;
      =     DB240.DBX  268.0;
      =     DB240.DBX  348.0;

      A     #RRel;
      A     M    102.3;
      =     DB240.DBX  108.0;

// -------------------------------------------------
// subphase transition
      L     #U.Seq.User.Real10;
      L     #U.Seq.SFM[10].Sp;
      <>R   ;
      O     #S2I.SFM10.I00;
      =     #xTmp;

      A     #xTmp;
      ON    DB145.DBX   26.4;
      =     M    103.1;

      A     #xTmp; // Tankwechsel
      JC    COMM;
      L     MW   118;
      L     -1;
      +I    ;
      T     MW   116;
      JU    COMM;

// subphase 3: Tank Change
A503: SET   ;
      L     #U.Seq.User.Real10;
      T     #U.Seq.SFM[10].Sp; // Current Tank

// -------------------------------------------------
// subphase timer & counter
      A     M    103.0;

// -------------------------------------------------
// subphase actuator
      A     M    103.3;

// -------------------------------------------------
// subphase transition
      AN    #S2I.SFM10.I00;
      AN    M    102.2;
      =     M    103.1;
      JU    COMM;
NETWORK
TITLE =phase 8: Push Out
//SFM   Use                                 Datatype        UoM
//----+-------------------------------------------------------------------------
// 00 : Watch Dog Time                      Duration        min
// 20 : Flow                                Value           l/h
// 41 : Amount                              Value           kg
X8:   SET   ;
// ---------------------------------------------------------------------------
// General CM evaluation
      CALL FC   140 (
           ChkType                  := 3,
           ChkOK                    := #ChkOK);

      AN    #ChkOK;
      S     M    120.3;

// Current Tank
      L     #U.Seq.User.Real10;
      T     #U.Seq.SFM[10].Sp;

// ---------------------------------------------------------------------------
// general functions
      L     #LineID;
      L     DB145.DBD  242;
      AW    ;
      L     #LineID;
      ==I   ;
      CLR   ;
      AN    M    121.2;
      A     M    102.3;
      =     #RRel;

// ---------------------------------------------------------------------------
// messages
// ---------------------------------------------------------------------------
// timer & counter

// ---------------------------------------------------------------------------
// pause timer
      AN    #ComSRC;
      ON    M    102.3;
      O     M    152.0;
      S     M    142.0;

      AN    M    102.3;
      O     M    150.7;
      S     M    140.7;

// ---------------------------------------------------------------------------
// communication
      A     M    102.0;
      =     DB145.DBX   29.1;

// ---------------------------------------------------------------------------
// control modules

// ---------------------------------------------------------------------------
// transition condition
      AN    #ComCIPDist;
      A     #SubStepMaxD;
      =     M    102.1;

// subphase evaluation
      L     MW   110;
      JL    A800;
      JU    COMM; // subphase  0:
      JU    A801; // subphase  1: Waiting
      JU    A802; // subphase  2: Active
      JU    A803; // subphase  3: Backwards
      JU    A804; // subphase  4: CIP Start
// ---------------------------------------------------------------------------
A800: SET   ;
      S     M    110.7; // Error unknown subphase
      JU    COMM;

// subphase 1: Waiting
A801: SET   ;
      A     M    103.3;
      =     DB145.DBX   26.3;
      =     DB145.DBX   26.0;
// -------------------------------------------------
// subphase timer & counter
      A     M    103.0;

// -------------------------------------------------
// subphase actuator
      A     M    103.3;

// -------------------------------------------------
// subphase transition
      SET   ;
      =     M    103.1;
      JU    COMM;

// subphase 2: Active
A802: SET   ;
      A     M    103.3;
      =     DB145.DBX   26.4;
      =     DB145.DBX   26.1;
      =     DB145.DBX  173.7; // CIP Ende

// -------------------------------------------------
// subphase timer & counter
      A     M    103.0;

// -------------------------------------------------
// subphase actuator

// -------------------------------------------------
// subphase transition
      SET   ;
      =     M    103.1;
      JU    COMM;

// subphase 3: Backwards
A803: SET   ;
      A     DB145.DBX  411.5;
      A     DB145.DBX   75.4;
      A     DB240.DBX  422.6;
      O     DB240.DBX  502.6;
      O     DB240.DBX  582.6;
      A     #ComSRC;
      A     M    103.3;
      =     DB145.DBX   26.1;

// -------------------------------------------------
// subphase timer & counter
      A     DB145.DBX  218.4;
      A     M    103.0;
      =     M    130.7; // Substep Time

// -------------------------------------------------
// subphase actuator
      A     #RRel;
      A     #ComCIPDist;
      A     M    103.3;
      =     DB145.DBX  173.6; // Req Common Drain

      A     #RRel;
      A     #ComCIPDist;
      A     #ComDistCIP1;
      A     M    103.3;
      =     DB240.DBX  428.0; // CIP Distribution 1

      A     #RRel;
      A     #ComCIPDist;
      A     #ComDistCIP2;
      A     M    103.3;
      =     DB240.DBX  508.0; // CIP Distribution 2

      A     #RRel;
      A     #ComCIPDist;
      A     #ComDistCIP3;
      A     M    103.3;
      =     DB240.DBX  588.0; // CIP Distribution 3

// -------------------------------------------------
// subphase transition
      A     M    150.7; // Substep Time Done
      AN    M    103.2;
      =     M    103.1;
      JU    COMM;

// subphase 4: CIP Start
A804: SET   ;
// CIP Distribution Start
      L     #U.Seq.SFM[18].Sp;
      L     1.000000e+000; // Auto select
      ==I   ;
      JCN   CIPb;
      L     MB   112;
      L     43;
      ==I   ;
      JC    N5sd;
      CALL FC   711 (
           StartType                := 6,
           Release                  := TRUE,
           CIPEqID                  := #iTmp);
      JU    Fin1;
N5sd: NOP   0;
      L     3095;
      T     #iTmp;
Fin1: NOP   0;

      L     0;
      L     #iTmp;
      ==I   ;
      JC    CIPb;
      ITD   ;
      DTR   ;
      T     #U.Seq.SFM[18].Sp; // CIP Distribution Start
CIPb: NOP   0;

//---
// CIP 1 Start
      L     #U.Seq.SFM[18].Sp;
      L     3.094000e+003; // CIP 1
      ==I   ;
      JCN   X8a;
      L     MD   124;
      T     DB502.DBD  156;
X8a:  NOP   0;

//---
// CIP 2 Start
      L     #U.Seq.SFM[18].Sp;
      L     3.095000e+003; // CIP 2
      ==I   ;
      JCN   X8b;
      L     MD   124;
      T     DB502.DBD  160;
X8b:  NOP   0;

//---
// CIP 3 Start
      L     #U.Seq.SFM[18].Sp;
      L     3.096000e+003; // CIP 3
      ==I   ;
      JCN   X8c;
      L     MD   124;
      T     DB502.DBD  164;
X8c:  NOP   0;

// -------------------------------------------------
// subphase timer & counter
      A     M    103.0;

// -------------------------------------------------
// subphase actuator
      A     M    103.3;

// -------------------------------------------------
// subphase transition
// CIP Distribution Ready
      A     #ComCIPDist;
      =     M    103.1;

      JU    COMM;


NETWORK
TITLE =phase 11: Postrinse
//SFM   Use                                 Datatype        UoM
//----+-------------------------------------------------------------------------
// 00 : Watch Dog Time                      Duration        min
// 20 : Flow                                Value           l/h
// 41 : Amount                              Value           kg
X11:  SET   ;
// ---------------------------------------------------------------------------
// General CM evaluation
      CALL FC   140 (
           ChkType                  := 3,
           ChkOK                    := #ChkOK);

      AN    #ChkOK;
      S     M    120.3;

// ---------------------------------------------------------------------------
// general functions
      AN    M    121.2;
      A     M    102.3;
      =     #RRel;

// ---------------------------------------------------------------------------
// messages
// ---------------------------------------------------------------------------
// timer & counter
      A     M    102.0;

// ---------------------------------------------------------------------------
// pause timer
// ---------------------------------------------------------------------------
// communication

// ---------------------------------------------------------------------------
// control modules
      A     M    102.3;

// ---------------------------------------------------------------------------
// transition condition
      A     #SubStepMaxD;
      =     M    102.1;

// subphase evaluation
      L     MW   110;
      JL    B100;
      JU    COMM; // subphase  0:
// ---------------------------------------------------------------------------
B100: SET   ;
      S     M    110.7; // Error unknown subphase
      JU    COMM;
NETWORK
TITLE =phase 19: Remove Filter Candles
//SFM   Use                                 Datatype        UoM
//----+-------------------------------------------------------------------------
// 00 : Watch Dog Time                      Duration        min
X19:  SET   ;
// ---------------------------------------------------------------------------
// General CM evaluation
      CALL FC   140 (
           ChkType                  := 3,
           ChkOK                    := #ChkOK);

      AN    #ChkOK;
      S     M    120.3;

// index evaluation: Confirm Connections
      CALL FC    45 (
           SFM                      := #U.Seq.SFM[24].Sp,
           Indexes                  := #S2I.SFM24);

// ---------------------------------------------------------------------------
// general functions
      AN    M    121.2;
      A     M    102.3;
      =     #RRel;

// ---------------------------------------------------------------------------
// messages
      A     #S2I.SFM24.I00; // Please Select
      JCN   x191;
      L     929; // Confirm to Continue
      T     MD    90;
x191: NOP   0;

// ---------------------------------------------------------------------------
// timer & counter
// ---------------------------------------------------------------------------
// pause timer
// ---------------------------------------------------------------------------
// communication
// ---------------------------------------------------------------------------
// control modules
// ---------------------------------------------------------------------------
// transition condition
      A     #S2I.SFM24.I01; // Yes
      A     DB141.DBX   66.2;
      A     M    120.6;
      =     M    102.1;

// subphase evaluation
      L     MW   110;
      JL    B900;
      JU    COMM; // subphase  0:
// ---------------------------------------------------------------------------
B900: SET   ;
      S     M    110.7; // Error unknown subphase
      JU    COMM;
NETWORK
TITLE =phase 20: Replace Filter Candles
//SFM   Use                                 Datatype        UoM
//----+-------------------------------------------------------------------------
// 00 : Watch Dog Time                      Duration        min
X20:  SET   ;
// ---------------------------------------------------------------------------
// General CM evaluation
      CALL FC   140 (
           ChkType                  := 3,
           ChkOK                    := #ChkOK);

      AN    #ChkOK;
      S     M    120.3;

// index evaluation: Confirm Connections
      CALL FC    45 (
           SFM                      := #U.Seq.SFM[24].Sp,
           Indexes                  := #S2I.SFM24);

// ---------------------------------------------------------------------------
// general functions
      AN    M    121.2;
      A     M    102.3;
      =     #RRel;

      A     #S2I.SFM24.I01; // Yes
      R     DB141.DBX   66.2;

// ---------------------------------------------------------------------------
// messages
      A     #S2I.SFM24.I00; // Please Select
      JCN   x201;
      L     929; // Confirm to Continue
      T     MD    90;
x201: NOP   0;

// ---------------------------------------------------------------------------
// timer & counter
// ---------------------------------------------------------------------------
// pause timer
// ---------------------------------------------------------------------------
// communication
// ---------------------------------------------------------------------------
// control modules
// ---------------------------------------------------------------------------
// transition condition
      A     #S2I.SFM24.I01; // Yes
      A     M    120.6;
      =     M    102.1;

// subphase evaluation
      L     MW   110;
      JL    C000;
      JU    COMM; // subphase  0:
// ---------------------------------------------------------------------------
C000: SET   ;
      S     M    110.7; // Error unknown subphase
      JU    COMM;
NETWORK
TITLE =phase 21: Prepare Line
//SFM   Use                                 Datatype        UoM
//----+-------------------------------------------------------------------------
// 00 : Watch Dog Time                      Duration        min
X21:  SET   ;
// ---------------------------------------------------------------------------
// General CM evaluation
      CALL FC   140 (
           ChkType                  := 3,
           ChkOK                    := #ChkOK);

      AN    #ChkOK;
      S     M    120.3;

// ---------------------------------------------------------------------------
// general functions
      AN    M    121.2;
      A     M    102.3;
      =     #RRel;

// ---------------------------------------------------------------------------
// messages
// ---------------------------------------------------------------------------
// timer & counter
      A     M    102.0;

// ---------------------------------------------------------------------------
// pause timer
// ---------------------------------------------------------------------------
// communication

// ---------------------------------------------------------------------------
// control modules
      A     M    102.3;

// ---------------------------------------------------------------------------
// transition condition
      A     #SubStepMaxD;
      =     M    102.1;

// subphase evaluation
      L     MW   110;
      JL    C100;
      JU    COMM; // subphase  0:
// ---------------------------------------------------------------------------
C100: SET   ;
      S     M    110.7; // Error unknown subphase
      JU    COMM;
NETWORK
TITLE =phase 22: Tank Selection
//SFM   Use                                 Datatype        UoM
//----+-------------------------------------------------------------------------
// 00 : Watch Dog Time                      Duration        min
X22:  SET   ;
// ---------------------------------------------------------------------------
// General CM evaluation
      CALL FC   140 (
           ChkType                  := 3,
           ChkOK                    := #ChkOK);

      AN    #ChkOK;
      S     M    120.3;

// ---------------------------------------------------------------------------
// general functions
      AN    M    121.2;
      A     M    102.3;
      =     #RRel;

// ---------------------------------------------------------------------------
// messages
      AN    #S2I.SFM11.I00; // Priority 1 Tank
      JCN   N901;
      L     919; // "Press Start to Continue"
      T     MD    90;
N901: NOP   0;

      A     #S2I.SFM11.I00;
      JCN   N902;
      L     906; // "Source not Selected"
      T     MD    90;
N902: NOP   0;

// ---------------------------------------------------------------------------
// timer & counter
      A     M    102.0;

// ---------------------------------------------------------------------------
// pause timer
// ---------------------------------------------------------------------------
// communication
      A     M    102.0;
      R     DB145.DBX   26.4;
// ---------------------------------------------------------------------------
// control modules
      A     M    102.3;

// ---------------------------------------------------------------------------
// transition condition
      A     M    120.6;
      AN    #S2I.SFM11.I00; // Priority 1
      =     M    102.1;

// subphase evaluation
      L     MW   110;
      JL    C200;
      JU    COMM; // subphase  0:
// ---------------------------------------------------------------------------
C200: SET   ;
      S     M    110.7; // Error unknown subphase
      JU    COMM;
NETWORK
TITLE =phase 30: CIP Active
//SFM   Use                                 Datatype        UoM
//----+-------------------------------------------------------------------------
// 00 : Watch Dog Time                      Duration        min
// 05 : Substep Time                        Duration        s
// 22 : Pump Speed                          Value           %
X30:  SET   ;
// ---------------------------------------------------------------------------
// General CM evaluation
      CALL FC   140 (
           ChkType                  := 3,
           ChkOK                    := #ChkOK);

      AN    #ChkOK;
      S     M    120.3;

// ---------------------------------------------------------------------------
// general functions
      AN    M    121.2;
      A     M    102.3;
      =     #RRel;

// ---------------------------------------------------------------------------
// messages
// ---------------------------------------------------------------------------
// timer & counter
      A     M    102.0;

// ---------------------------------------------------------------------------
// pause timer
      ON    M    102.3;
      O     M    150.4;
      S     M    140.4; // Substep Time

// ---------------------------------------------------------------------------
// communication

// ---------------------------------------------------------------------------
// control modules
      A     M    102.3;

// ---------------------------------------------------------------------------
// transition condition
      A     #SubStepMaxD;
      =     M    102.1;

// ---------------------------------------------------------------------------
// ---------------------------------------------------------------------------
// subphase repeat function
//      A     #SubStepMax
//      JCN  Y30
//      L     1
//      T     "SOSubStepNew"
//Y30:  SET

// subphase evaluation
      L     MW   110;
      JL    D000;
      JU    COMM; // subphase  0:
      JU    D001; // subphase  1: Standby
      JU    D002; // subphase  2: Active
      JU    D003; // subphase  3: Expulse
// ---------------------------------------------------------------------------
D000: SET   ;
      S     M    110.7; // Error unknown subphase
      JU    COMM;

// subphase 1: Standby
D001: SET   ;

// -------------------------------------------------
// subphase timer & counter
      A     M    103.0;

// -------------------------------------------------
// subphase actuator
      A     M    103.3;

// -------------------------------------------------
// subphase transition
      CLR   ;
      =     M    103.1;
      JU    COMM;

// subphase 2: Active
D002: SET   ;

// -------------------------------------------------
// subphase timer & counter
      A     M    103.0;

// -------------------------------------------------
// subphase actuator
      A     M    103.3;

// -------------------------------------------------
// subphase transition
      CLR   ;
      =     M    103.1;
      JU    COMM;

// subphase 3: Expulse
D003: SET   ;

// -------------------------------------------------
// subphase timer & counter
      A     M    103.0;

// -------------------------------------------------
// subphase actuator
      A     M    103.3;

// -------------------------------------------------
// subphase transition
      CLR   ;
      =     M    103.1;
      JU    COMM;
NETWORK
TITLE =phase 31: CIP Start
//SFM   Use                                 Datatype        UoM
//----+-------------------------------------------------------------------------
// 00 : Watch Dog Time                      Duration        min
X31:  SET   ;

// ---------------------------------------------------------------------------
// General CM evaluation
      CALL FC   140 (
           ChkType                  := 3,
           ChkOK                    := #ChkOK);

      AN    #ChkOK;
      S     M    120.3;

// ---------------------------------------------------------------------------
// general functions
      AN    M    121.2;
      A     M    102.3;
      =     #RRel;

// ---------------------------------------------------------------------------
// messages
// ---------------------------------------------------------------------------
// timer & counter
// ---------------------------------------------------------------------------
// pause timer
// ---------------------------------------------------------------------------
// communication

// ---------------------------------------------------------------------------
// control modules


// ---------------------------------------------------------------------------
// transition condition
      A     #SubStepMaxD;
      =     M    102.1;

// ---------------------------------------------------------------------------
// ---------------------------------------------------------------------------
// subphase repeat function
//      A     #SubStepMax
//      JCN  Y31
//      L     1
//      T     "SOSubStepNew"
//Y31:  SET

// subphase evaluation
      L     MW   110;
      JL    D100;
      JU    COMM; // subphase  0:
      JU    D101; // subphase  1: Wait For CIP
      JU    D102; // subphase  2: Wait For Partner
// ---------------------------------------------------------------------------
D100: SET   ;
      S     M    110.7; // Error unknown subphase
      JU    COMM;

// subphase 1: Wait For CIP
D101: SET   ;

// CIP  Start
      L     0;
      T     #iTmp;

      L     #U.Seq.SFM[18].Sp;
      L     1.000000e+000; // Auto select
      ==I   ;
      JCN   CIPa;


      L     MB   112;
      L     43;
      ==I   ;
      JC    U43S;
      CALL FC   711 (
           StartType                := 7,// Priority CIP 2, 1, 3 (Anlagen)
           Release                  := TRUE,
           CIPEqID                  := #iTmp);
      JU    NU43;
U43S: L     3092; // KEG Only CIP 2
      T     #iTmp;
NU43: NOP   0;


      L     0;
      L     #iTmp;
      ==I   ;
      JC    CIPa;
      ITD   ;
      DTR   ;
      T     #U.Seq.SFM[18].Sp; // CIP  Start
CIPa: NOP   0;

//---
// CIP 1 Start
      L     #U.Seq.SFM[18].Sp;
      L     3.091000e+003; // CIP 1
      ==I   ;
      JCN   X31a;
      L     MD   124;
      T     DB502.DBD    0;
      T     DB502.DBD  156;
X31a: NOP   0;

//---
// CIP 2 Start
      L     #U.Seq.SFM[18].Sp;
      L     3.092000e+003; // CIP 2
      ==I   ;

      JCN   X31b;
      L     MD   124;
      T     DB502.DBD    4;
      T     DB502.DBD  160;
X31b: NOP   0;

//---
// CIP 3 Start
      L     #U.Seq.SFM[18].Sp;
      L     3.093000e+003; // CIP 3
      ==I   ;
      JCN   X31c;
      L     MD   124;
      T     DB502.DBD    8;
      T     DB502.DBD  164;
X31c: NOP   0;

// -------------------------------------------------
// subphase timer & counter

// -------------------------------------------------
// subphase actuator

// -------------------------------------------------
// subphase transition
// CIP Ready
      A     #ComCIP;
      A     DB145.DBX  123.5;
      A     DB145.DBX  120.0;
// CIP Distribution Ready
      A     #ComCIPDist;
      A     DB145.DBX  411.5;
      A     DB145.DBX  408.0;
      =     M    103.1;
      JU    COMM;

// subphase 2: Wait For Partner
D102: SET   ;

      A     M    103.0;
      =     DB145.DBX   29.4; // Request Packaging Plant

// -------------------------------------------------
// subphase timer & counter

// -------------------------------------------------
// subphase actuator

// -------------------------------------------------
// subphase transition
      A     DB145.DBX  459.4;
      =     M    103.1;
      JU    COMM;
NETWORK
TITLE =phase 32: CIP Prerun
//SFM   Use                                 Datatype        UoM
//----+-------------------------------------------------------------------------
// 00 : Watch Dog Time                      Duration        min
// 01 : Step Time                           Duration        min
// 04 : Delay Level                         Duration        s
// 15 : Amount                              Value           m3
// 17 : Level                               Value           l
// 22 : Agitator Speed                      Value           %
// 27 : CIP Prerun                          Enumeration     min
// 28 : CIP Return                          Enumeration     min
// 29 : CIP Pump Speed                      Value           %
// 34 : CIP Prerun Flow                     Value           m3/h
// 35 : CIP Prerun Pressure                 Value           bar
// 37 : CIP Pump Mode                       Enumeration     min
X32:  SET   ;
// ---------------------------------------------------------------------------
// General CM evaluation
      CALL FC   140 (
           ChkType                  := 3,
           ChkOK                    := #ChkOK);

      AN    #ChkOK;
      S     M    120.3;

// ---------------------------------------------------------------------------
// index evaluation: CIP Prerun
      CALL FC    45 (
           SFM                      := #U.Seq.SFM[27].Sp,
           Indexes                  := #S2I.SFM27);

// ---------------------------------------------------------------------------
// index evaluation: CIP Return
      CALL FC    45 (
           SFM                      := #U.Seq.SFM[28].Sp,
           Indexes                  := #S2I.SFM28);

// ---------------------------------------------------------------------------
// index evaluation: CIP Pump Mode
      CALL FC    45 (
           SFM                      := #U.Seq.SFM[37].Sp,
           Indexes                  := #S2I.SFM37);

// ---------------------------------------------------------------------------
// general functions
      AN    M    121.2;
      A     M    102.3;
      =     #RRel;

// Get Pushout Amount

      A     M    102.2;
      JCN   N321;
      L     #U.Seq.Prop.Val10;
      L     #U.Seq.SFM[15].Sp;
      +R    ;
      T     #U.Seq.SFM[15].Sp;
N321: NOP   0;

// CIP Unit
      AN    #ComCIP;
      ON    DB145.DBX  123.4;
      ON    DB145.DBX  123.5;
      JCN   x321;
      R     #RRel;
      L     949; // CIP Not Ready!
      T     MD    90;
x321: NOP   0;

// CIP Distribution Unit
      AN    #ComCIPDist;
      ON    DB145.DBX  411.4;
      ON    DB145.DBX  411.5;
      JCN   x322;
      R     #RRel;
      L     949; // CIP Not Ready!
      T     MD    90;
x322: NOP   0;

// Partner Unit
      AN    #ComDST;
      ON    DB145.DBX  459.4;
      ON    DB145.DBX  459.5;
      JCN   x323;
      R     #RRel;
      L     903; // Partner Unit Not Ready!
      T     MD    90;
x323: NOP   0;

// CIP Signals ---
      CALL FC   716 (
           StepOnSFMSP              := #U.Seq.SFM[26].Sp,
           EmptySig                 := DB145.DBX  458.5,
           EmptyLevel               := TRUE,
           CIPPumpRun               := DB145.DBX  124.3,
           CIPReady                 := DB145.DBX  123.5,
           Empty                    := #Empty,
           TransCondOK              := M    102.1,
           RRel                     := #RRel);

      A     DB145.DBX  124.3;
      A     M    102.3;
      =     DB145.DBX   29.2;

// ---------------------------------------------------------------------------
// messages
// ---------------------------------------------------------------------------
// timer & counter
// Done in "CIPUnitC"

// ---------------------------------------------------------------------------
// communication
// Active, Prerun & Return
      A     M    102.0;
      =     DB145.DBX  171.4;
      =     DB145.DBX  172.6;
      =     DB145.DBX  172.7;

// Run Release
      A     #RRel;
      =     DB145.DBX  171.5;

// Prerun Pump
      A     DB145.DBX  459.5;
      A     DB145.DBX  459.6;
      A     DB145.DBX  172.6;
      AN    #S2I.SFM37.I00;
      A     #RRel;
      =     DB145.DBX  173.3;

// Return Pump
      AN    #Empty;
      A     #RRel;
      =     DB145.DBX  173.4;
      =     DB145.DBX   29.3;

// ---------------------------------------------------------------------------
// control modules (Own CM's)
      A     #ComCIP1;
      A     M    102.3;
      =     DB240.DBX  428.0;

      A     #ComCIP2;
      A     M    102.3;
      =     DB240.DBX  508.0;

      A     #ComCIP3;
      A     M    102.3;
      =     DB240.DBX  588.0;

// Trap Filter
      A     #S2I.SFM14.I01; // Yes
      A     M    102.3;
      CLR   ;
      =     DB240.DBX  188.0;
      =     DB240.DBX  348.0;

      A     #S2I.SFM14.I01; // Yes
      A     M    102.3;
      =     DB240.DBX  268.0;

// ---------------------------------------------------------------------------
// transition condition
//      A     #SubStepMaxD
//      =     "SOPD"

// subphase evaluation
      L     MW   110;
      JL    D200;
      JU    COMM; // subphase  0:
// ---------------------------------------------------------------------------
D200: SET   ;
      S     M    110.7; // Error unknown subphase
      JU    COMM;
NETWORK
TITLE =phase 33: CIP Return
//SFM   Use                                 Datatype        UoM
//----+-------------------------------------------------------------------------
// 00 : Watch Dog Time                      Duration        min
// 01 : Step Time                           Duration        min
// 04 : Delay Level                         Duration        s
// 06 : Delay Switchpoint                   Duration        s
// 15 : Amount                              Value           m3
// 17 : Level                               Value           l
// 22 : Agitator Speed                      Value           %
// 26 : CIP Step On Condition               Enumeration     min
// 27 : CIP Prerun                          Enumeration     min
// 28 : CIP Return                          Enumeration     min
// 29 : CIP Pump Speed                      Value           %
// 30 : CIP Return Temperature              Value           °C
// 32 : CIP Return Conductivity             Value           mS
// 34 : CIP Prerun Flow                     Value           m3/h
// 35 : CIP Prerun Pressure                 Value           bar
// 37 : CIP Pump Mode                       Enumeration     min
X33:  SET   ;
// ---------------------------------------------------------------------------
// General CM evaluation
      CALL FC   140 (
           ChkType                  := 3,
           ChkOK                    := #ChkOK);

      AN    #ChkOK;
      S     M    120.3;

// ---------------------------------------------------------------------------
// index evaluation: CIP Step On Condition
      CALL FC    45 (
           SFM                      := #U.Seq.SFM[26].Sp,
           Indexes                  := #S2I.SFM26);

// ---------------------------------------------------------------------------
// index evaluation: CIP Prerun
      CALL FC    45 (
           SFM                      := #U.Seq.SFM[27].Sp,
           Indexes                  := #S2I.SFM27);

// ---------------------------------------------------------------------------
// index evaluation: CIP Return
      CALL FC    45 (
           SFM                      := #U.Seq.SFM[28].Sp,
           Indexes                  := #S2I.SFM28);

// ---------------------------------------------------------------------------
// index evaluation: CIP Pump Mode
      CALL FC    45 (
           SFM                      := #U.Seq.SFM[37].Sp,
           Indexes                  := #S2I.SFM37);

// ---------------------------------------------------------------------------
// general functions
      AN    M    121.2;
      A     M    102.3;
      =     #RRel;

// ---------------------------------------------------------------------------
// messages
// CIP Unit
      AN    #ComCIP;
      ON    DB145.DBX  123.4;
      ON    DB145.DBX  123.5;
      JCN   x331;
      R     #RRel;
      L     949; // CIP Not Ready!
      T     MD    90;
x331: NOP   0;

// CIP Distribution Unit
      AN    #ComCIPDist;
      ON    DB145.DBX  411.4;
      ON    DB145.DBX  411.5;
      JCN   x332;
      R     #RRel;
      L     949; // CIP Partner Not Ready!
      T     MD    90;
x332: NOP   0;

// Partner Unit
      AN    #ComDST;
      ON    DB145.DBX  459.4;
      ON    DB145.DBX  459.5;
      JCN   x333;
      R     #RRel;
      L     903; // Partner Unit Not Ready!
      T     MD    90;
x333: NOP   0;

// CIP Signals ---
      CALL FC   716 (
           StepOnSFMSP              := #U.Seq.SFM[26].Sp,
           EmptySig                 := DB145.DBX  458.5,
           EmptyLevel               := TRUE,
           CIPPumpRun               := DB145.DBX  124.3,
           CIPReady                 := DB145.DBX  123.5,
           Empty                    := #Empty,
           TransCondOK              := M    102.1,
           RRel                     := #RRel);


      A     DB145.DBX  124.3;
      A     M    102.3;
      =     DB145.DBX   29.2;

// ---------------------------------------------------------------------------
// timer & counter
// Done in "CIPUnitC"

// ---------------------------------------------------------------------------
// communication
// Active, Prerun & Return
      A     M    102.0;
      =     DB145.DBX  171.4;
      =     DB145.DBX  172.6;
      =     DB145.DBX  172.7;

// Run Release
      A     #RRel;
      =     DB145.DBX  171.5;

// Prerun Pump
      A     DB145.DBX  459.5;
      A     DB145.DBX  459.6;
      A     DB145.DBX  172.6;
      AN    #S2I.SFM37.I00;
      A     #RRel;
      =     DB145.DBX  173.3;

// Return Pump
      AN    #Empty;
      A     #RRel;
      =     DB145.DBX  173.4;
      =     DB145.DBX   29.3;

// Bypass Valve
      A     M    102.3;
      =     DB145.DBX  173.5;

// ---------------------------------------------------------------------------
// control modules (Own CM's)
      A     #ComCIP1;
      A     M    102.3;
      =     DB240.DBX  428.0;

      A     #ComCIP2;
      A     M    102.3;
      =     DB240.DBX  508.0;

      A     #ComCIP3;
      A     M    102.3;
      =     DB240.DBX  588.0;

// Trap Filter
      A     #S2I.SFM14.I01; // Yes
      A     M    102.3;
      CLR   ;
      =     DB240.DBX  188.0;
      =     DB240.DBX  348.0;

      A     #S2I.SFM14.I01; // Yes
      A     M    102.3;
      =     DB240.DBX  268.0;

// Bypass Valve Used in CIP Distribution
//      A     "SOPA"
//      =     "c04ActD".RV1_T13.ACo

//      A     "SOPH"
//      =     "c04ActD".T13_RR1.ACo

// ---------------------------------------------------------------------------
// transition condition
//      A     #SubStepMaxD
//      =     "SOPD"

// subphase evaluation
      L     MW   110;
      JL    D300;
      JU    COMM; // subphase  0:
// ---------------------------------------------------------------------------
D300: SET   ;
      S     M    110.7; // Error unknown subphase
      JU    COMM;
NETWORK
TITLE =phase 34: CIP Rinsing
//SFM   Use                                 Datatype        UoM
//----+-------------------------------------------------------------------------
// 00 : Watch Dog Time                      Duration        min
// 01 : Step Time                           Duration        min
// 05 : Substep Time                        Duration        s
// 06 : Delay Switchpoint                   Duration        s
// 15 : Amount                              Value           m3
// 27 : CIP Prerun                          Enumeration     min
// 28 : CIP Return                          Enumeration     min
// 29 : CIP Pump Speed                      Value           %
// 30 : CIP Return Temperature              Value           °C
// 32 : CIP Return Conductivity             Value           mS
// 34 : CIP Prerun Flow                     Value           m3/h
// 35 : CIP Prerun Pressure                 Value           bar
// 37 : CIP Pump Mode                       Enumeration     min
// 59 : Interval Counter                    Value           No.
X34:  SET   ;
// ---------------------------------------------------------------------------
// General CM evaluation
      CALL FC   140 (
           ChkType                  := 3,
           ChkOK                    := #ChkOK);

      AN    #ChkOK;
      S     M    120.3;

// ---------------------------------------------------------------------------
// index evaluation: CIP Prerun
      CALL FC    45 (
           SFM                      := #U.Seq.SFM[27].Sp,
           Indexes                  := #S2I.SFM27);

// ---------------------------------------------------------------------------
// index evaluation: CIP Return
      CALL FC    45 (
           SFM                      := #U.Seq.SFM[28].Sp,
           Indexes                  := #S2I.SFM28);

// ---------------------------------------------------------------------------
// index evaluation: CIP Pump Mode
      CALL FC    45 (
           SFM                      := #U.Seq.SFM[37].Sp,
           Indexes                  := #S2I.SFM37);

// ---------------------------------------------------------------------------
// general functions
      AN    M    121.2;
      A     M    102.3;
      =     #RRel;

// CIP Unit
      AN    #ComCIP;
      ON    DB145.DBX  123.4;
      ON    DB145.DBX  123.5;
      JCN   x341;
      R     #RRel;
      L     949; // CIP Not Ready!
      T     MD    90;
x341: NOP   0;

// CIP Distribution Unit
      AN    #ComCIPDist;
      ON    DB145.DBX  411.4;
      ON    DB145.DBX  411.5;
      JCN   x342;
      R     #RRel;
      L     949; // CIP Partner Not Ready!
      T     MD    90;
x342: NOP   0;

// Partner Unit
      AN    #ComDST;
      ON    DB145.DBX  459.4;
      ON    DB145.DBX  459.5;
      JCN   x343;
      R     #RRel;
      L     903; // Partner Unit Not Ready!
      T     MD    90;
x343: NOP   0;

// CIP Signals ---
      CALL FC   716 (
           StepOnSFMSP              := #U.Seq.SFM[26].Sp,
           EmptySig                 := DB145.DBX  458.5,
           EmptyLevel               := TRUE,
           CIPPumpRun               := DB145.DBX  124.3,
           CIPReady                 := DB145.DBX  123.5,
           Empty                    := #Empty,
           TransCondOK              := M    102.1,
           RRel                     := #RRel);

      A     DB145.DBX  124.3;
      A     M    102.3;
      =     DB145.DBX   29.2;



// ---------------------------------------------------------------------------
// messages
// ---------------------------------------------------------------------------
// timer & counter
// Done in "CIPUnitC"

// ---------------------------------------------------------------------------
// pause timer
      ON    M    102.3;
      O     M    150.0;
      S     M    140.0; // Step Time

      ON    M    102.3;
      O     M    150.5;
      S     M    140.5; // Delay Switchpoint

// ---------------------------------------------------------------------------
// communication
// Active, Prerun & Return
      A     M    102.0;
      =     DB145.DBX  171.4;
      =     DB145.DBX  172.7;
      =     DB145.DBX  172.6;

// Run Release
      A     #RRel;
      =     DB145.DBX  171.5;

// Prerun Pump
      A     DB145.DBX  459.5;
      A     DB145.DBX  459.6;
      A     DB145.DBX  172.6;
      AN    #S2I.SFM37.I00;
      A     #RRel;
      =     DB145.DBX  173.3;

// Return Pump
      AN    #Empty;
      A     #RRel;
      =     DB145.DBX  173.4;
      =     DB145.DBX   29.3;

// Mit Ablauf
      AN    M    157.2;
      A     M    102.0;
      =     DB145.DBX   29.5;

// ---------------------------------------------------------------------------
// control modules (Own CM's)
      A     #ComCIP1;
      A     M    102.3;
      =     DB240.DBX  428.0;

      A     #ComCIP2;
      A     M    102.3;
      =     DB240.DBX  508.0;

      A     #ComCIP3;
      A     M    102.3;
      =     DB240.DBX  588.0;

// Trap Filter
      A     #S2I.SFM14.I01; // Yes
      A     M    102.3;
      CLR   ;
      =     DB240.DBX  188.0;
      =     DB240.DBX  348.0;

      A     #S2I.SFM14.I01; // Yes
      A     M    102.3;
      =     DB240.DBX  268.0;

// ---------------------------------------------------------------------------
// transition condition
//      A     #SubStepMaxD
//      =     "SOPD"

// ---------------------------------------------------------------------------
// ---------------------------------------------------------------------------
// subphase repeat function
      A     #SubStepMax;
      JCN   Y34;
      L     1;
      T     MW   116;
Y34:  SET   ;

      A     #SubStepMax;
      AN    M    103.0;
      JCN   Y34a;
      L     #U.Seq.SFM[59].Val; // Increment Interval Counter
      L     1.000000e+000;
      +R    ;
      T     #U.Seq.SFM[59].Val;
Y34a: SET   ;
      A     M    102.2;
      ON    M    102.0;
      JCN   IntR; // Reset Interval Counter at Start and End Of Phase
      L     0.000000e+000;
      T     #U.Seq.SFM[59].Val;
IntR: NOP   0;

// subphase evaluation
      L     MW   110;
      JL    D400;
      JU    COMM; // subphase  0:
      JU    D401; // subphase  1: Pause
      JU    D402; // subphase  2: Main
      JU    D403; // subphase  3: Expulse
      JU    D404; // subphase  4: Seat Lift
      JU    D400; // subphase  5:
      JU    D406; // subphase  6: Shaft Rinse
      JU    D407; // subphase  7: Drain
// ---------------------------------------------------------------------------
D400: SET   ;
      S     M    110.7; // Error unknown subphase
      JU    COMM;

// subphase 1: Pause
D401: SET   ;

      A     M    103.0;
      R     DB145.DBX  173.3;

// -------------------------------------------------
// subphase timer & counter
      A     M    103.0;
      =     M    130.4; // Substep Time
// -------------------------------------------------
// subphase actuator

// -------------------------------------------------
// subphase transition
      A     M    150.3; // Delay Level
      A     M    130.3;
      O     M    150.4; // Substep Time Done
      =     M    103.1;
      JU    COMM;

// subphase 2: Main
D402: SET   ;

// -------------------------------------------------
// subphase timer & counter
      A     M    103.0;
      =     M    130.4; // Substep Time

// -------------------------------------------------
// subphase actuator
      A     M    103.3;


// -------------------------------------------------
// subphase transition
      A     M    150.4; // Substep Time Done
      =     M    103.1;
      JU    COMM;

// subphase 3: Expulse
D403: SET   ;

// -------------------------------------------------
// subphase timer & counter
      A     M    103.0;

// -------------------------------------------------
// subphase actuator
      A     M    103.3;

// -------------------------------------------------
// subphase transition
      CLR   ;
      =     M    103.1;
      JU    COMM;

// subphase 4: Seat Lift
D404: SET   ;

// -------------------------------------------------
// subphase timer & counter
      A     M    103.0;

// -------------------------------------------------
// subphase actuator
      A     M    103.3;

// -------------------------------------------------
// subphase transition
      SET   ;
      =     M    103.1;
      JU    COMM;

// subphase 6: Shaft Rinse
D406: SET   ;

// -------------------------------------------------
// subphase timer & counter
      A     M    103.0;
      =     M    130.4; // Substep Time

// -------------------------------------------------
// subphase actuator
      A     M    103.3;
      =     DB240.DBX  668.0;

// -------------------------------------------------
// subphase transition
      A     M    150.4; // Substep Time Done
      O     M    157.2; // Interval Counter Done
      =     M    103.1;
      JU    COMM;

// subphase 7: Drain
D407: SET   ;

// -------------------------------------------------
// subphase timer & counter
      A     M    103.0;
      =     M    130.4; // Substep Time

// -------------------------------------------------
// subphase actuator
      A     M    103.3;
      R     DB145.DBX  173.6; // Req Drain RV1_RS
      R     DB145.DBX   29.6; // Req Common Drain
      R     DB2990.DBX  268.0;

// -------------------------------------------------
// subphase transition
      A     M    150.4; // Substep Time Done
      O     M    157.2; // Interval Counter Done
      =     M    103.1;
      JU    COMM;
NETWORK
TITLE =phase 35: CIP Emptying
//SFM   Use                                 Datatype        UoM
//----+-------------------------------------------------------------------------
// 00 : Watch Dog Time                      Duration        min
// 04 : Delay Empty                         Duration        s
// 17 : Level                               Value           l
// 22 : Agitator Speed                      Value           %
// 26 : Step On Empty                       Enumeration     min
// 28 : CIP Return                          Enumeration     min
X35:  SET   ;
// ---------------------------------------------------------------------------
// General CM evaluation
      CALL FC   140 (
           ChkType                  := 3,
           ChkOK                    := #ChkOK);

      AN    #ChkOK;
      S     M    120.3;

// ---------------------------------------------------------------------------
// index evaluation: Step On Empty
      CALL FC    45 (
           SFM                      := #U.Seq.SFM[26].Sp,
           Indexes                  := #S2I.SFM26);

// ---------------------------------------------------------------------------
// index evaluation: CIP Return
      CALL FC    45 (
           SFM                      := #U.Seq.SFM[28].Sp,
           Indexes                  := #S2I.SFM28);

// ---------------------------------------------------------------------------
// general functions
      AN    M    121.2;
      A     M    102.3;
      =     #RRel;

// ---------------------------------------------------------------------------
// messages
// CIP Unit
      AN    #ComCIP;
      ON    DB145.DBX  123.4;
      ON    DB145.DBX  123.5;
      JCN   x351;
      R     #RRel;
      L     949; // CIP Not Ready!
      T     MD    90;
x351: NOP   0;

// CIP Distribution Unit
      AN    #ComCIPDist;
      ON    DB145.DBX  411.4;
      ON    DB145.DBX  411.5;
      JCN   x352;
      R     #RRel;
      L     949; // CIP Partner Not Ready!
      T     MD    90;
x352: NOP   0;

// Partner Unit
      AN    #ComDST;
      ON    DB145.DBX  459.4;
      ON    DB145.DBX  459.5;
      JCN   x353;
      R     #RRel;
      L     903; // Partner Unit Not Ready!
      T     MD    90;
x353: NOP   0;

// CIP Signals ---
      CALL FC   716 (
           StepOnSFMSP              := #U.Seq.SFM[26].Sp,
           EmptySig                 := DB145.DBX  458.5,
           EmptyLevel               := TRUE,
           CIPPumpRun               := DB145.DBX  124.3,
           CIPReady                 := DB145.DBX  123.5,
           Empty                    := #Empty,
           TransCondOK              := M    102.1,
           RRel                     := #RRel);

// ---------------------------------------------------------------------------
// timer & counter
// Done in "CIPUnitC"

// ---------------------------------------------------------------------------
// communication
// Active, Prerun & Return
      A     M    102.0;
      =     DB145.DBX  171.4;
      =     DB145.DBX  172.7;
      CLR   ;
      =     DB145.DBX  172.6;

// Run Release
      A     #RRel;
      =     DB145.DBX  171.5;

